LIN {X 0,Y 277.298,Z 529.083,A -85,B 0,C 180,E1 -17480.317,E2 -17480.317} C_VEL
LIN {X 0,Y 276.413,Z 532.07,A -85,B 0,C 180,E1 -17482.419,E2 -17482.419} C_VEL
LIN {X 0,Y 275.927,Z 533.774,A -85,B 0,C 180,E1 -17484.049,E2 -17484.049} C_VEL
LIN {X 0,Y 275.323,Z 535.445,A -85,B 0,C 180,E1 -17486.689,E2 -17486.689} C_VEL
LIN {X 0,Y 274.975,Z 535.726,A -85,B 0,C 180,E1 -17489.654,E2 -17489.654} C_VEL
LIN {X 0,Y 274.909,Z 534.486,A -85,B 0,C 180,E1 -17492.47,E2 -17492.47} C_VEL
LIN {X 0,Y 275.167,Z 531.808,A -85,B 0,C 180,E1 -17495.18,E2 -17495.18} C_VEL
LIN {X 0,Y 275.645,Z 527.856,A -85,B 0,C 180,E1 -17497.774,E2 -17497.774} C_VEL
LIN {X 0,Y 276.168,Z 522.667,A -85,B 0,C 180,E1 -17500.227,E2 -17500.227} C_VEL
LIN {X 0,Y 277.018,Z 516.038,A -85,B 0,C 180,E1 -17502.627,E2 -17502.627} C_VEL
LIN {X 0,Y 278.075,Z 507.892,A -85,B 0,C 180,E1 -17504.952,E2 -17504.952} C_VEL
LIN {X 0,Y 279.237,Z 499.452,A -85,B 0,C 180,E1 -17506.876,E2 -17506.876} C_VEL
LIN {X 0,Y 280.566,Z 489.56,A -85,B 0,C 180,E1 -17508.718,E2 -17508.718} C_VEL
LIN {X 0,Y 282.003,Z 478.351,A -85,B 0,C 180,E1 -17510.385,E2 -17510.385} C_VEL
LIN {X 0,Y 283.262,Z 466.509,A -85,B 0,C 180,E1 -17511.785,E2 -17511.785} C_VEL
LIN {X 0,Y 281.61,Z 454.332,A -85,B 0,C 180,E1 -17513.056,E2 -17513.056} C_VEL
LIN {X 0,Y 279.109,Z 440.408,A -85,B 0,C 180,E1 -17514.219,E2 -17514.219} C_VEL
LIN {X 0,Y 276.812,Z 428.738,A -85,B 0,C 180,E1 -17514.965,E2 -17514.965} C_VEL
LIN {X 0,Y 277.178,Z 422.689,A -85,B 0,C 180,E1 -17518.68,E2 -17518.68} C_VEL
LIN {X 0,Y 277.552,Z 416.666,A -85,B 0,C 180,E1 -17522.404,E2 -17522.404} C_VEL
LIN {X 0,Y 277.936,Z 410.649,A -85,B 0,C 180,E1 -17526.132,E2 -17526.132} C_VEL
LIN {X 0,Y 277.632,Z 407.009,A -85,B 0,C 180,E1 -17528.463,E2 -17528.463} C_VEL
LIN {X 0,Y 277.421,Z 405.931,A -85,B 0,C 180,E1 -17529.224,E2 -17529.224} C_VEL
LIN {X 0,Y 277.446,Z 405.925,A -85,B 0,C 180,E1 -17534.275,E2 -17534.275} C_VEL
LIN {X 0,Y 277.436,Z 405.93,A -85,B 0,C 180,E1 -17538.305,E2 -17538.305} C_VEL
LIN {X 0,Y 277.571,Z 405.911,A -85,B 0,C 180,E1 -17541.259,E2 -17541.259} C_VEL
LIN {X 0,Y 277.511,Z 405.956,A -85,B 0,C 180,E1 -17544.73,E2 -17544.73} C_VEL
LIN {X 0,Y 278.433,Z 410.139,A -85,B 0,C 180,E1 -17548.55,E2 -17548.55} C_VEL
LIN {X 0,Y 278.074,Z 413.616,A -85,B 0,C 180,E1 -17551.445,E2 -17551.445} C_VEL
LIN {X 0,Y 277.432,Z 418.956,A -85,B 0,C 180,E1 -17555.812,E2 -17555.812} C_VEL
LIN {X 0,Y 277.034,Z 422.666,A -85,B 0,C 180,E1 -17558.752,E2 -17558.752} C_VEL
LIN {X 0,Y 276.611,Z 427.071,A -85,B 0,C 180,E1 -17562.189,E2 -17562.189} C_VEL
LIN {X 0,Y 279.223,Z 439.231,A -85,B 0,C 180,E1 -17563.089,E2 -17563.089} C_VEL
LIN {X 0,Y 281.351,Z 451.494,A -85,B 0,C 180,E1 -17564.277,E2 -17564.277} C_VEL
LIN {X 0,Y 282.477,Z 460.237,A -85,B 0,C 180,E1 -17565.325,E2 -17565.325} C_VEL
LIN {X 0,Y 281.293,Z 470.488,A -85,B 0,C 180,E1 -17566.694,E2 -17566.694} C_VEL
LIN {X 0,Y 280.009,Z 480.226,A -85,B 0,C 180,E1 -17568.349,E2 -17568.349} C_VEL
LIN {X 0,Y 278.753,Z 489.099,A -85,B 0,C 180,E1 -17570.28,E2 -17570.28} C_VEL
LIN {X 0,Y 277.708,Z 496.37,A -85,B 0,C 180,E1 -17572.305,E2 -17572.305} C_VEL
LIN {X 0,Y 277.006,Z 501.3,A -85,B 0,C 180,E1 -17574.026,E2 -17574.026} C_VEL
LIN {X 0,Y 276.268,Z 506.386,A -85,B 0,C 180,E1 -17576.303,E2 -17576.303} C_VEL
LIN {X 0,Y 275.857,Z 509.379,A -85,B 0,C 180,E1 -17578.116,E2 -17578.116} C_VEL
LIN {X 0,Y 275.478,Z 512.199,A -85,B 0,C 180,E1 -17580.675,E2 -17580.675} C_VEL
LIN {X 0,Y 275.366,Z 513.344,A -85,B 0,C 180,E1 -17582.624,E2 -17582.624} C_VEL
LIN {X 0,Y 275.417,Z 513.666,A -85,B 0,C 180,E1 -17584.147,E2 -17584.147} C_VEL
LIN {X 0,Y 275.596,Z 513.368,A -85,B 0,C 180,E1 -17585.906,E2 -17585.906} C_VEL
LIN {X 0,Y 275.986,Z 512.222,A -85,B 0,C 180,E1 -17587.87,E2 -17587.87} C_VEL
LIN {X 0,Y 276.777,Z 509.44,A -85,B 0,C 180,E1 -17590.38,E2 -17590.38} C_VEL
LIN {X 0,Y 277.754,Z 505.303,A -85,B 0,C 180,E1 -17592.796,E2 -17592.796} C_VEL
LIN {X 0,Y 279.084,Z 499.564,A -85,B 0,C 180,E1 -17595.163,E2 -17595.163} C_VEL
LIN {X 0,Y 280.373,Z 493.538,A -85,B 0,C 180,E1 -17597.076,E2 -17597.076} C_VEL
LIN {X 0,Y 282.213,Z 485.156,A -85,B 0,C 180,E1 -17599.13,E2 -17599.13} C_VEL
LIN {X 0,Y 283.843,Z 477.123,A -85,B 0,C 180,E1 -17600.686,E2 -17600.686} C_VEL
LIN {X 0,Y 285.699,Z 466.304,A -85,B 0,C 180,E1 -17602.339,E2 -17602.339} C_VEL
LIN {X 0,Y 285.302,Z 460.121,A -85,B 0,C 180,E1 -17603.232,E2 -17603.232} C_VEL
LIN {X 0,Y 283.597,Z 449.539,A -85,B 0,C 180,E1 -17604.624,E2 -17604.624} C_VEL
LIN {X 0,Y 281.033,Z 439.046,A -85,B 0,C 180,E1 -17605.814,E2 -17605.814} C_VEL
LIN {X 0,Y 277.584,Z 428.375,A -85,B 0,C 180,E1 -17606.913,E2 -17606.913} C_VEL
LIN {X 0,Y 278.098,Z 423.388,A -85,B 0,C 180,E1 -17611.305,E2 -17611.305} C_VEL
LIN {X 0,Y 278.623,Z 419.781,A -85,B 0,C 180,E1 -17614.609,E2 -17614.609} C_VEL
LIN {X 0,Y 278.806,Z 416.478,A -85,B 0,C 180,E1 -17617.784,E2 -17617.784} C_VEL
LIN {X 0,Y 278.619,Z 413.529,A -85,B 0,C 180,E1 -17620.858,E2 -17620.858} C_VEL
LIN {X 0,Y 278.253,Z 410.854,A -85,B 0,C 180,E1 -17623.87,E2 -17623.87} C_VEL
LIN {X 0,Y 277.652,Z 407.251,A -85,B 0,C 180,E1 -17628.317,E2 -17628.317} C_VEL
LIN {X 0,Y 277.514,Z 405.917,A -85,B 0,C 180,E1 -17630.153,E2 -17630.153} C_VEL
LIN {X 0,Y 277.631,Z 405.905,A -85,B 0,C 180,E1 -17632.729,E2 -17632.729} C_VEL
LIN {X 0,Y 277.669,Z 405.898,A -85,B 0,C 180,E1 -17636.986,E2 -17636.986} C_VEL
LIN {X 0,Y 277.204,Z 405.963,A -85,B 0,C 180,E1 -17638.198,E2 -17638.198} C_VEL
LIN {X 0,Y 275.718,Z 406.15,A -85,B 0,C 180,E1 -17639.389,E2 -17639.389} C_VEL
LIN {X 0,Y 271.004,Z 406.729,A -85,B 0,C 180,E1 -17642.602,E2 -17642.602} C_VEL
LIN {X 0,Y 270.557,Z 406.778,A -85,B 0,C 180,E1 -17643.444,E2 -17643.444} C_VEL
LIN {X 0,Y 270.591,Z 406.776,A -85,B 0,C 180,E1 -17647.462,E2 -17647.462} C_VEL
LIN {X 0,Y 270.422,Z 406.798,A -85,B 0,C 180,E1 -17650.482,E2 -17650.482} C_VEL
LIN {X 0,Y 270.383,Z 406.8,A -85,B 0,C 180,E1 -17655.066,E2 -17655.066} C_VEL
LIN {X 0,Y 270.308,Z 406.815,A -85,B 0,C 180,E1 -17659.756,E2 -17659.756} C_VEL
LIN {X 0,Y 270.261,Z 406.814,A -85,B 0,C 180,E1 -17664.587,E2 -17664.587} C_VEL
LIN {X 0,Y 270.255,Z 406.817,A -85,B 0,C 180,E1 -17667.911,E2 -17667.911} C_VEL
LIN {X 0,Y 270.168,Z 406.831,A -85,B 0,C 180,E1 -17671.351,E2 -17671.351} C_VEL
LIN {X 0,Y 270.265,Z 407.011,A -85,B 0,C 180,E1 -17675.618,E2 -17675.618} C_VEL
LIN {X 0,Y 270.839,Z 409.72,A -85,B 0,C 180,E1 -17678.886,E2 -17678.886} C_VEL
LIN {X 0,Y 271.495,Z 412.982,A -85,B 0,C 180,E1 -17682.303,E2 -17682.303} C_VEL
LIN {X 0,Y 272.353,Z 416.818,A -85,B 0,C 180,E1 -17685.841,E2 -17685.841} C_VEL
LIN {X 0,Y 273.431,Z 422.485,A -85,B 0,C 180,E1 -17690.453,E2 -17690.453} C_VEL
LIN {X 0,Y 274.584,Z 428.793,A -85,B 0,C 180,E1 -17694.99,E2 -17694.99} C_VEL
LIN {X 0,Y 274.945,Z 431.299,A -85,B 0,C 180,E1 -17696.667,E2 -17696.667} C_VEL
LIN {X 0,Y 274.499,Z 434.05,A -85,B 0,C 180,E1 -17698.351,E2 -17698.351} C_VEL
LIN {X 0,Y 272.629,Z 441.637,A -85,B 0,C 180,E1 -17702.68,E2 -17702.68} C_VEL
LIN {X 0,Y 275.821,Z 455.459,A -85,B 0,C 180,E1 -17703.791,E2 -17703.791} C_VEL
LIN {X 0,Y 277.753,Z 468.394,A -85,B 0,C 180,E1 -17705.038,E2 -17705.038} C_VEL
LIN {X 0,Y 278.418,Z 478.611,A -85,B 0,C 180,E1 -17706.183,E2 -17706.183} C_VEL
LIN {X 0,Y 278.3,Z 489.099,A -85,B 0,C 180,E1 -17707.549,E2 -17707.549} C_VEL
LIN {X 0,Y 276.287,Z 499.847,A -85,B 0,C 180,E1 -17709.142,E2 -17709.142} C_VEL
LIN {X 0,Y 274.262,Z 509.481,A -85,B 0,C 180,E1 -17710.934,E2 -17710.934} C_VEL
LIN {X 0,Y 272.621,Z 517.98,A -85,B 0,C 180,E1 -17712.936,E2 -17712.936} C_VEL
LIN {X 0,Y 271.197,Z 524.971,A -85,B 0,C 180,E1 -17714.984,E2 -17714.984} C_VEL
LIN {X 0,Y 269.826,Z 531.068,A -85,B 0,C 180,E1 -17717.213,E2 -17717.213} C_VEL
LIN {X 0,Y 269.001,Z 535.877,A -85,B 0,C 180,E1 -17719.466,E2 -17719.466} C_VEL
LIN {X 0,Y 268.404,Z 540.987,A -85,B 0,C 180,E1 -17722.481,E2 -17722.481} C_VEL
LIN {X 0,Y 268.227,Z 544.686,A -85,B 0,C 180,E1 -17724.668,E2 -17724.668} C_VEL
LIN {X 0,Y 268.229,Z 547.519,A -85,B 0,C 180,E1 -17727,E2 -17727} C_VEL
LIN {X 0,Y 268.234,Z 548.777,A -85,B 0,C 180,E1 -17728.502,E2 -17728.502} C_VEL
LIN {X 0,Y 268.229,Z 549.619,A -85,B 0,C 180,E1 -17730.003,E2 -17730.003} C_VEL
LIN {X 0,Y 268.227,Z 550.004,A -85,B 0,C 180,E1 -17731.505,E2 -17731.505} C_VEL
LIN {X 0,Y 268.208,Z 549.981,A -85,B 0,C 180,E1 -17733.007,E2 -17733.007} C_VEL
LIN {X 0,Y 268.175,Z 549.223,A -85,B 0,C 180,E1 -17735.212,E2 -17735.212} C_VEL
LIN {X 0,Y 268.456,Z 547.489,A -85,B 0,C 180,E1 -17737.525,E2 -17737.525} C_VEL
LIN {X 0,Y 269.002,Z 544.845,A -85,B 0,C 180,E1 -17739.78,E2 -17739.78} C_VEL
LIN {X 0,Y 269.892,Z 541.2,A -85,B 0,C 180,E1 -17742.027,E2 -17742.027} C_VEL
LIN {X 0,Y 271.146,Z 536.498,A -85,B 0,C 180,E1 -17744.258,E2 -17744.258} C_VEL
LIN {X 0,Y 273.181,Z 529.479,A -85,B 0,C 180,E1 -17746.826,E2 -17746.826} C_VEL
LIN {X 0,Y 275.243,Z 521.489,A -85,B 0,C 180,E1 -17749.133,E2 -17749.133} C_VEL
LIN {X 0,Y 277.76,Z 512.629,A -85,B 0,C 180,E1 -17751.137,E2 -17751.137} C_VEL
LIN {X 0,Y 280.193,Z 503.213,A -85,B 0,C 180,E1 -17752.882,E2 -17752.882} C_VEL
LIN {X 0,Y 282.704,Z 492.898,A -85,B 0,C 180,E1 -17754.415,E2 -17754.415} C_VEL
LIN {X 0,Y 283.337,Z 483.957,A -85,B 0,C 180,E1 -17755.679,E2 -17755.679} C_VEL
LIN {X 0,Y 283.169,Z 472.199,A -85,B 0,C 180,E1 -17757.171,E2 -17757.171} C_VEL
LIN {X 0,Y 281.892,Z 460.18,A -85,B 0,C 180,E1 -17758.598,E2 -17758.598} C_VEL
LIN {X 0,Y 279.764,Z 449.124,A -85,B 0,C 180,E1 -17759.832,E2 -17759.832} C_VEL
LIN {X 0,Y 275.311,Z 434.987,A -85,B 0,C 180,E1 -17761.559,E2 -17761.559} C_VEL
LIN {X 0,Y 275.347,Z 431.758,A -85,B 0,C 180,E1 -17762.616,E2 -17762.616} C_VEL
LIN {X 0,Y 274.35,Z 426.033,A -85,B 0,C 180,E1 -17764.94,E2 -17764.94} C_VEL
LIN {X 0,Y 272.837,Z 419.7,A -85,B 0,C 180,E1 -17768.189,E2 -17768.189} C_VEL
LIN {X 0,Y 271.854,Z 414.556,A -85,B 0,C 180,E1 -17771.434,E2 -17771.434} C_VEL
LIN {X 0,Y 271.327,Z 410.842,A -85,B 0,C 180,E1 -17774.379,E2 -17774.379} C_VEL
LIN {X 0,Y 271.135,Z 409.615,A -85,B 0,C 180,E1 -17775.584,E2 -17775.584} C_VEL
LIN {X 0,Y 270.16,Z 406.826,A -85,B 0,C 180,E1 -17779.798,E2 -17779.798} C_VEL
LIN {X 0,Y 270.231,Z 406.823,A -85,B 0,C 180,E1 -17783.733,E2 -17783.733} C_VEL
LIN {X 0,Y 270.21,Z 406.826,A -85,B 0,C 180,E1 -17786.893,E2 -17786.893} C_VEL
LIN {X 0,Y 270.167,Z 406.831,A -85,B 0,C 180,E1 -17790.379,E2 -17790.379} C_VEL
LIN {X 0,Y 270.222,Z 406.993,A -85,B 0,C 180,E1 -17794.587,E2 -17794.587} C_VEL
LIN {X 0,Y 270.989,Z 409.489,A -85,B 0,C 180,E1 -17799.016,E2 -17799.016} C_VEL
LIN {X 0,Y 271.946,Z 412.845,A -85,B 0,C 180,E1 -17803.484,E2 -17803.484} C_VEL
LIN {X 0,Y 272.58,Z 415.707,A -85,B 0,C 180,E1 -17806.582,E2 -17806.582} C_VEL
LIN {X 0,Y 273.223,Z 418.787,A -85,B 0,C 180,E1 -17809.626,E2 -17809.626} C_VEL
LIN {X 0,Y 273.835,Z 422.113,A -85,B 0,C 180,E1 -17812.627,E2 -17812.627} C_VEL
LIN {X 0,Y 274.033,Z 423.867,A -85,B 0,C 180,E1 -17814.111,E2 -17814.111} C_VEL
LIN {X 0,Y 273.835,Z 426.752,A -85,B 0,C 180,E1 -17816.321,E2 -17816.321} C_VEL
LIN {X 0,Y 273.103,Z 430.671,A -85,B 0,C 180,E1 -17819.123,E2 -17819.123} C_VEL
LIN {X 0,Y 274.489,Z 434.354,A -85,B 0,C 180,E1 -17819.67,E2 -17819.67} C_VEL
LIN {X 0,Y 279.094,Z 445.971,A -85,B 0,C 180,E1 -17821.442,E2 -17821.442} C_VEL
LIN {X 0,Y 282.187,Z 456.631,A -85,B 0,C 180,E1 -17823.038,E2 -17823.038} C_VEL
LIN {X 0,Y 284.054,Z 466.96,A -85,B 0,C 180,E1 -17824.576,E2 -17824.576} C_VEL
LIN {X 0,Y 284.871,Z 476.125,A -85,B 0,C 180,E1 -17826.018,E2 -17826.018} C_VEL
LIN {X 0,Y 283.66,Z 482.538,A -85,B 0,C 180,E1 -17826.89,E2 -17826.89} C_VEL
LIN {X 0,Y 281.037,Z 493.447,A -85,B 0,C 180,E1 -17828.629,E2 -17828.629} C_VEL
LIN {X 0,Y 278.405,Z 503.103,A -85,B 0,C 180,E1 -17830.555,E2 -17830.555} C_VEL
LIN {X 0,Y 275.732,Z 512.265,A -85,B 0,C 180,E1 -17832.886,E2 -17832.886} C_VEL
LIN {X 0,Y 273.512,Z 519.589,A -85,B 0,C 180,E1 -17835.27,E2 -17835.27} C_VEL
LIN {X 0,Y 271.838,Z 525.028,A -85,B 0,C 180,E1 -17837.528,E2 -17837.528} C_VEL
LIN {X 0,Y 270.512,Z 529.16,A -85,B 0,C 180,E1 -17839.739,E2 -17839.739} C_VEL
LIN {X 0,Y 269.713,Z 531.578,A -85,B 0,C 180,E1 -17841.395,E2 -17841.395} C_VEL
LIN {X 0,Y 268.897,Z 534.132,A -85,B 0,C 180,E1 -17843.821,E2 -17843.821} C_VEL
LIN {X 0,Y 268.188,Z 535.826,A -85,B 0,C 180,E1 -17846.998,E2 -17846.998} C_VEL
LIN {X 0,Y 267.867,Z 535.803,A -85,B 0,C 180,E1 -17850.02,E2 -17850.02} C_VEL
LIN {X 0,Y 267.814,Z 534.241,A -85,B 0,C 180,E1 -17852.883,E2 -17852.883} C_VEL
LIN {X 0,Y 268.158,Z 531.305,A -85,B 0,C 180,E1 -17855.659,E2 -17855.659} C_VEL
LIN {X 0,Y 268.653,Z 527.044,A -85,B 0,C 180,E1 -17858.294,E2 -17858.294} C_VEL
LIN {X 0,Y 269.213,Z 521.598,A -85,B 0,C 180,E1 -17860.79,E2 -17860.79} C_VEL
LIN {X 0,Y 270.184,Z 514.647,A -85,B 0,C 180,E1 -17863.25,E2 -17863.25} C_VEL
LIN {X 0,Y 271.271,Z 506.161,A -85,B 0,C 180,E1 -17865.609,E2 -17865.609} C_VEL
LIN {X 0,Y 272.617,Z 497.03,A -85,B 0,C 180,E1 -17867.643,E2 -17867.643} C_VEL
LIN {X 0,Y 273.992,Z 486.938,A -85,B 0,C 180,E1 -17869.454,E2 -17869.454} C_VEL
LIN {X 0,Y 275.506,Z 475.358,A -85,B 0,C 180,E1 -17871.124,E2 -17871.124} C_VEL
LIN {X 0,Y 276.317,Z 466.857,A -85,B 0,C 180,E1 -17872.124,E2 -17872.124} C_VEL
LIN {X 0,Y 274.612,Z 454.825,A -85,B 0,C 180,E1 -17873.419,E2 -17873.419} C_VEL
LIN {X 0,Y 272.214,Z 441.187,A -85,B 0,C 180,E1 -17874.587,E2 -17874.587} C_VEL
LIN {X 0,Y 269.81,Z 428.871,A -85,B 0,C 180,E1 -17875.412,E2 -17875.412} C_VEL
LIN {X 0,Y 270.177,Z 422.923,A -85,B 0,C 180,E1 -17879.138,E2 -17879.138} C_VEL
LIN {X 0,Y 270.575,Z 416.82,A -85,B 0,C 180,E1 -17882.961,E2 -17882.961} C_VEL
LIN {X 0,Y 270.937,Z 411.551,A -85,B 0,C 180,E1 -17886.29,E2 -17886.29} C_VEL
LIN {X 0,Y 270.579,Z 407.891,A -85,B 0,C 180,E1 -17888.673,E2 -17888.673} C_VEL
LIN {X 0,Y 270.389,Z 406.806,A -85,B 0,C 180,E1 -17889.534,E2 -17889.534} C_VEL
LIN {X 0,Y 270.384,Z 406.805,A -85,B 0,C 180,E1 -17894.096,E2 -17894.096} C_VEL
LIN {X 0,Y 270.399,Z 406.805,A -85,B 0,C 180,E1 -17897.996,E2 -17897.996} C_VEL
LIN {X 0,Y 270.528,Z 406.789,A -85,B 0,C 180,E1 -17901.029,E2 -17901.029} C_VEL
LIN {X 0,Y 270.491,Z 406.884,A -85,B 0,C 180,E1 -17904.405,E2 -17904.405} C_VEL
LIN {X 0,Y 271.42,Z 411.271,A -85,B 0,C 180,E1 -17908.513,E2 -17908.513} C_VEL
LIN {X 0,Y 271.039,Z 414.754,A -85,B 0,C 180,E1 -17911.482,E2 -17911.482} C_VEL
LIN {X 0,Y 270.383,Z 420.16,A -85,B 0,C 180,E1 -17915.964,E2 -17915.964} C_VEL
LIN {X 0,Y 269.944,Z 423.882,A -85,B 0,C 180,E1 -17918.983,E2 -17918.983} C_VEL
LIN {X 0,Y 269.606,Z 427.292,A -85,B 0,C 180,E1 -17921.699,E2 -17921.699} C_VEL
LIN {X 0,Y 272.374,Z 439.904,A -85,B 0,C 180,E1 -17922.666,E2 -17922.666} C_VEL
LIN {X 0,Y 274.441,Z 452.083,A -85,B 0,C 180,E1 -17923.888,E2 -17923.888} C_VEL
LIN {X 0,Y 275.56,Z 460.769,A -85,B 0,C 180,E1 -17924.961,E2 -17924.961} C_VEL
LIN {X 0,Y 274.392,Z 470.924,A -85,B 0,C 180,E1 -17926.36,E2 -17926.36} C_VEL
LIN {X 0,Y 273.132,Z 480.269,A -85,B 0,C 180,E1 -17927.981,E2 -17927.981} C_VEL
LIN {X 0,Y 271.764,Z 489.503,A -85,B 0,C 180,E1 -17930.035,E2 -17930.035} C_VEL
LIN {X 0,Y 270.685,Z 496.763,A -85,B 0,C 180,E1 -17932.111,E2 -17932.111} C_VEL
LIN {X 0,Y 269.809,Z 502.654,A -85,B 0,C 180,E1 -17934.262,E2 -17934.262} C_VEL
LIN {X 0,Y 269.165,Z 507.019,A -85,B 0,C 180,E1 -17936.347,E2 -17936.347} C_VEL
LIN {X 0,Y 268.632,Z 510.88,A -85,B 0,C 180,E1 -17938.942,E2 -17938.942} C_VEL
LIN {X 0,Y 268.449,Z 512.229,A -85,B 0,C 180,E1 -17940.239,E2 -17940.239} C_VEL
LIN {X 0,Y 268.297,Z 513.881,A -85,B 0,C 180,E1 -17943.047,E2 -17943.047} C_VEL
LIN {X 0,Y 268.494,Z 513.869,A -85,B 0,C 180,E1 -17945.764,E2 -17945.764} C_VEL
LIN {X 0,Y 269.033,Z 512.393,A -85,B 0,C 180,E1 -17948.401,E2 -17948.401} C_VEL
LIN {X 0,Y 269.919,Z 509.449,A -85,B 0,C 180,E1 -17950.968,E2 -17950.968} C_VEL
LIN {X 0,Y 270.986,Z 505.129,A -85,B 0,C 180,E1 -17953.434,E2 -17953.434} C_VEL
LIN {X 0,Y 272.447,Z 499.247,A -85,B 0,C 180,E1 -17955.855,E2 -17955.855} C_VEL
LIN {X 0,Y 274.042,Z 492.168,A -85,B 0,C 180,E1 -17958.043,E2 -17958.043} C_VEL
LIN {X 0,Y 275.787,Z 484.67,A -85,B 0,C 180,E1 -17959.856,E2 -17959.856} C_VEL
LIN {X 0,Y 277.731,Z 475.146,A -85,B 0,C 180,E1 -17961.664,E2 -17961.664} C_VEL
LIN {X 0,Y 279.109,Z 467.553,A -85,B 0,C 180,E1 -17962.821,E2 -17962.821} C_VEL
LIN {X 0,Y 278.725,Z 461.209,A -85,B 0,C 180,E1 -17963.784,E2 -17963.784} C_VEL
LIN {X 0,Y 276.91,Z 449.799,A -85,B 0,C 180,E1 -17965.343,E2 -17965.343} C_VEL
LIN {X 0,Y 274.172,Z 439.214,A -85,B 0,C 180,E1 -17966.618,E2 -17966.618} C_VEL
LIN {X 0,Y 270.673,Z 428.605,A -85,B 0,C 180,E1 -17967.786,E2 -17967.786} C_VEL
LIN {X 0,Y 271.276,Z 423.758,A -85,B 0,C 180,E1 -17972.204,E2 -17972.204} C_VEL
LIN {X 0,Y 271.768,Z 420.211,A -85,B 0,C 180,E1 -17975.559,E2 -17975.559} C_VEL
LIN {X 0,Y 271.879,Z 417.045,A -85,B 0,C 180,E1 -17978.784,E2 -17978.784} C_VEL
LIN {X 0,Y 271.554,Z 414.216,A -85,B 0,C 180,E1 -17981.907,E2 -17981.907} C_VEL
LIN {X 0,Y 271.19,Z 411.64,A -85,B 0,C 180,E1 -17984.981,E2 -17984.981} C_VEL
LIN {X 0,Y 270.813,Z 409.274,A -85,B 0,C 180,E1 -17988.018,E2 -17988.018} C_VEL
LIN {X 0,Y 270.559,Z 406.784,A -85,B 0,C 180,E1 -17991.599,E2 -17991.599} C_VEL
LIN {X 0,Y 270.525,Z 406.786,A -85,B 0,C 180,E1 -17994.036,E2 -17994.036} C_VEL
LIN {X 0,Y 270.773,Z 406.752,A -85,B 0,C 180,E1 -17998.513,E2 -17998.513} C_VEL
LIN {X 0,Y 270.773,Z 406.752,A -85,B 0,C 180,E1 -18001.488,E2 -18001.488} C_VEL
LIN {X 0,Y 270.557,Z 406.778,A -85,B 0,C 180,E1 -18003.444,E2 -18003.444} C_VEL
LIN {X 0,Y 269.762,Z 406.883,A -85,B 0,C 180,E1 -18004.687,E2 -18004.687} C_VEL
LIN {X 0,Y 266.937,Z 407.228,A -85,B 0,C 180,E1 -18006.716,E2 -18006.716} C_VEL
LIN {X 0,Y 263.778,Z 407.624,A -85,B 0,C 180,E1 -18009.209,E2 -18009.209} C_VEL
LIN {X 0,Y 263.41,Z 407.668,A -85,B 0,C 180,E1 -18010.071,E2 -18010.071} C_VEL
LIN {X 0,Y 263.289,Z 407.689,A -85,B 0,C 180,E1 -18013.901,E2 -18013.901} C_VEL
LIN {X 0,Y 263.256,Z 407.694,A -85,B 0,C 180,E1 -18017.078,E2 -18017.078} C_VEL
LIN {X 0,Y 263.25,Z 407.689,A -85,B 0,C 180,E1 -18020.882,E2 -18020.882} C_VEL
LIN {X 0,Y 263.194,Z 407.698,A -85,B 0,C 180,E1 -18025.293,E2 -18025.293} C_VEL
LIN {X 0,Y 263.163,Z 407.703,A -85,B 0,C 180,E1 -18028.732,E2 -18028.732} C_VEL
LIN {X 0,Y 263.176,Z 407.772,A -85,B 0,C 180,E1 -18033.651,E2 -18033.651} C_VEL
LIN {X 0,Y 263.72,Z 410.183,A -85,B 0,C 180,E1 -18036.927,E2 -18036.927} C_VEL
LIN {X 0,Y 264.197,Z 412.514,A -85,B 0,C 180,E1 -18039.676,E2 -18039.676} C_VEL
LIN {X 0,Y 265.217,Z 417.077,A -85,B 0,C 180,E1 -18044.324,E2 -18044.324} C_VEL
LIN {X 0,Y 266.153,Z 422.073,A -85,B 0,C 180,E1 -18048.695,E2 -18048.695} C_VEL
LIN {X 0,Y 267.063,Z 427.304,A -85,B 0,C 180,E1 -18052.757,E2 -18052.757} C_VEL
LIN {X 0,Y 268.009,Z 432.703,A -85,B 0,C 180,E1 -18056.591,E2 -18056.591} C_VEL
LIN {X 0,Y 267.502,Z 435.448,A -85,B 0,C 180,E1 -18058.306,E2 -18058.306} C_VEL
LIN {X 0,Y 265.935,Z 441.367,A -85,B 0,C 180,E1 -18061.783,E2 -18061.783} C_VEL
LIN {X 0,Y 269.287,Z 455.509,A -85,B 0,C 180,E1 -18063.018,E2 -18063.018} C_VEL
LIN {X 0,Y 271.088,Z 467.636,A -85,B 0,C 180,E1 -18064.242,E2 -18064.242} C_VEL
LIN {X 0,Y 271.871,Z 479.08,A -85,B 0,C 180,E1 -18065.573,E2 -18065.573} C_VEL
LIN {X 0,Y 271.717,Z 489.368,A -85,B 0,C 180,E1 -18066.974,E2 -18066.974} C_VEL
LIN {X 0,Y 269.652,Z 499.994,A -85,B 0,C 180,E1 -18068.604,E2 -18068.604} C_VEL
LIN {X 0,Y 267.548,Z 509.532,A -85,B 0,C 180,E1 -18070.436,E2 -18070.436} C_VEL
LIN {X 0,Y 266.008,Z 516.933,A -85,B 0,C 180,E1 -18072.215,E2 -18072.215} C_VEL
LIN {X 0,Y 264.302,Z 524.829,A -85,B 0,C 180,E1 -18074.583,E2 -18074.583} C_VEL
LIN {X 0,Y 262.874,Z 530.874,A -85,B 0,C 180,E1 -18076.869,E2 -18076.869} C_VEL
LIN {X 0,Y 261.981,Z 535.641,A -85,B 0,C 180,E1 -18079.18,E2 -18079.18} C_VEL
LIN {X 0,Y 261.244,Z 541.848,A -85,B 0,C 180,E1 -18083.05,E2 -18083.05} C_VEL
LIN {X 0,Y 261.096,Z 545.371,A -85,B 0,C 180,E1 -18085.372,E2 -18085.372} C_VEL
LIN {X 0,Y 261.138,Z 547.124,A -85,B 0,C 180,E1 -18086.918,E2 -18086.918} C_VEL
LIN {X 0,Y 261.16,Z 548.424,A -85,B 0,C 180,E1 -18088.461,E2 -18088.461} C_VEL
LIN {X 0,Y 261.154,Z 549.313,A -85,B 0,C 180,E1 -18090.003,E2 -18090.003} C_VEL
LIN {X 0,Y 261.152,Z 549.783,A -85,B 0,C 180,E1 -18091.545,E2 -18091.545} C_VEL
LIN {X 0,Y 261.119,Z 549.805,A -85,B 0,C 180,E1 -18093.089,E2 -18093.089} C_VEL
LIN {X 0,Y 261.157,Z 548.667,A -85,B 0,C 180,E1 -18096.183,E2 -18096.183} C_VEL
LIN {X 0,Y 261.39,Z 547.487,A -85,B 0,C 180,E1 -18097.729,E2 -18097.729} C_VEL
LIN {X 0,Y 262.272,Z 543.865,A -85,B 0,C 180,E1 -18100.815,E2 -18100.815} C_VEL
LIN {X 0,Y 263.313,Z 540,A -85,B 0,C 180,E1 -18103.116,E2 -18103.116} C_VEL
LIN {X 0,Y 264.84,Z 535.031,A -85,B 0,C 180,E1 -18105.392,E2 -18105.392} C_VEL
LIN {X 0,Y 266.764,Z 528.835,A -85,B 0,C 180,E1 -18107.639,E2 -18107.639} C_VEL
LIN {X 0,Y 268.868,Z 521.254,A -85,B 0,C 180,E1 -18109.868,E2 -18109.868} C_VEL
LIN {X 0,Y 271.741,Z 511.878,A -85,B 0,C 180,E1 -18112.028,E2 -18112.028} C_VEL
LIN {X 0,Y 274.357,Z 502.363,A -85,B 0,C 180,E1 -18113.797,E2 -18113.797} C_VEL
LIN {X 0,Y 276.582,Z 493.196,A -85,B 0,C 180,E1 -18115.193,E2 -18115.193} C_VEL
LIN {X 0,Y 277.288,Z 482.326,A -85,B 0,C 180,E1 -18116.784,E2 -18116.784} C_VEL
LIN {X 0,Y 277.127,Z 471.099,A -85,B 0,C 180,E1 -18118.264,E2 -18118.264} C_VEL
LIN {X 0,Y 275.58,Z 458.104,A -85,B 0,C 180,E1 -18119.877,E2 -18119.877} C_VEL
LIN {X 0,Y 274.082,Z 450.681,A -85,B 0,C 180,E1 -18120.781,E2 -18120.781} C_VEL
LIN {X 0,Y 270.401,Z 438.698,A -85,B 0,C 180,E1 -18122.316,E2 -18122.316} C_VEL
LIN {X 0,Y 269.117,Z 434.948,A -85,B 0,C 180,E1 -18122.874,E2 -18122.874} C_VEL
LIN {X 0,Y 268.202,Z 429.316,A -85,B 0,C 180,E1 -18125.207,E2 -18125.207} C_VEL
LIN {X 0,Y 266.466,Z 421.675,A -85,B 0,C 180,E1 -18129.275,E2 -18129.275} C_VEL
LIN {X 0,Y 265.665,Z 417.352,A -85,B 0,C 180,E1 -18132.206,E2 -18132.206} C_VEL
LIN {X 0,Y 265.327,Z 414.721,A -85,B 0,C 180,E1 -18134.341,E2 -18134.341} C_VEL
LIN {X 0,Y 264.884,Z 412.911,A -85,B 0,C 180,E1 -18136.382,E2 -18136.382} C_VEL
LIN {X 0,Y 263.985,Z 410.296,A -85,B 0,C 180,E1 -18140.286,E2 -18140.286} C_VEL
LIN {X 0,Y 263.476,Z 408.985,A -85,B 0,C 180,E1 -18144.067,E2 -18144.067} C_VEL
LIN {X 0,Y 263.329,Z 408.727,A -85,B 0,C 180,E1 -18147.738,E2 -18147.738} C_VEL
LIN {X 0,Y 263.52,Z 409.254,A -85,B 0,C 180,E1 -18151.659,E2 -18151.659} C_VEL
LIN {X 0,Y 263.94,Z 410.363,A -85,B 0,C 180,E1 -18154.872,E2 -18154.872} C_VEL
LIN {X 0,Y 264.433,Z 412.145,A -85,B 0,C 180,E1 -18158.474,E2 -18158.474} C_VEL
LIN {X 0,Y 265.242,Z 414.97,A -85,B 0,C 180,E1 -18162.537,E2 -18162.537} C_VEL
LIN {X 0,Y 265.922,Z 418.079,A -85,B 0,C 180,E1 -18166.239,E2 -18166.239} C_VEL
LIN {X 0,Y 266.843,Z 422.657,A -85,B 0,C 180,E1 -18170.907,E2 -18170.907} C_VEL
LIN {X 0,Y 267.322,Z 426.049,A -85,B 0,C 180,E1 -18173.963,E2 -18173.963} C_VEL
LIN {X 0,Y 267.236,Z 427.907,A -85,B 0,C 180,E1 -18175.474,E2 -18175.474} C_VEL
LIN {X 0,Y 266.75,Z 431.106,A -85,B 0,C 180,E1 -18177.763,E2 -18177.763} C_VEL
LIN {X 0,Y 268.131,Z 434.652,A -85,B 0,C 180,E1 -18178.317,E2 -18178.317} C_VEL
LIN {X 0,Y 271.755,Z 443.605,A -85,B 0,C 180,E1 -18179.814,E2 -18179.814} C_VEL
LIN {X 0,Y 275.434,Z 454.99,A -85,B 0,C 180,E1 -18181.665,E2 -18181.665} C_VEL
LIN {X 0,Y 277.81,Z 466.705,A -85,B 0,C 180,E1 -18183.542,E2 -18183.542} C_VEL
LIN {X 0,Y 278.723,Z 477.886,A -85,B 0,C 180,E1 -18185.364,E2 -18185.364} C_VEL
LIN {X 0,Y 277.675,Z 483.123,A -85,B 0,C 180,E1 -18186.117,E2 -18186.117} C_VEL
LIN {X 0,Y 274.868,Z 493.984,A -85,B 0,C 180,E1 -18187.899,E2 -18187.899} C_VEL
LIN {X 0,Y 272.058,Z 503.705,A -85,B 0,C 180,E1 -18189.899,E2 -18189.899} C_VEL
LIN {X 0,Y 269.451,Z 512.01,A -85,B 0,C 180,E1 -18192.043,E2 -18192.043} C_VEL
LIN {X 0,Y 267.138,Z 519.414,A -85,B 0,C 180,E1 -18194.472,E2 -18194.472} C_VEL
LIN {X 0,Y 264.928,Z 525.857,A -85,B 0,C 180,E1 -18197.246,E2 -18197.246} C_VEL
LIN {X 0,Y 263.553,Z 529.77,A -85,B 0,C 180,E1 -18199.47,E2 -18199.47} C_VEL
LIN {X 0,Y 262.381,Z 533.06,A -85,B 0,C 180,E1 -18202.024,E2 -18202.024} C_VEL
LIN {X 0,Y 261.721,Z 534.821,A -85,B 0,C 180,E1 -18204.071,E2 -18204.071} C_VEL
LIN {X 0,Y 261.359,Z 535.625,A -85,B 0,C 180,E1 -18205.482,E2 -18205.482} C_VEL
LIN {X 0,Y 261.041,Z 536.176,A -85,B 0,C 180,E1 -18207.315,E2 -18207.315} C_VEL
LIN {X 0,Y 260.738,Z 535.796,A -85,B 0,C 180,E1 -18210.393,E2 -18210.393} C_VEL
LIN {X 0,Y 260.778,Z 533.956,A -85,B 0,C 180,E1 -18213.333,E2 -18213.333} C_VEL
LIN {X 0,Y 261.181,Z 530.498,A -85,B 0,C 180,E1 -18216.297,E2 -18216.297} C_VEL
LIN {X 0,Y 261.667,Z 526.206,A -85,B 0,C 180,E1 -18218.836,E2 -18218.836} C_VEL
LIN {X 0,Y 262.338,Z 520.426,A -85,B 0,C 180,E1 -18221.396,E2 -18221.396} C_VEL
LIN {X 0,Y 263.339,Z 513.023,A -85,B 0,C 180,E1 -18223.938,E2 -18223.938} C_VEL
LIN {X 0,Y 264.554,Z 504.259,A -85,B 0,C 180,E1 -18226.311,E2 -18226.311} C_VEL
LIN {X 0,Y 266.138,Z 493.764,A -85,B 0,C 180,E1 -18228.561,E2 -18228.561} C_VEL
LIN {X 0,Y 267.64,Z 482.547,A -85,B 0,C 180,E1 -18230.46,E2 -18230.46} C_VEL
LIN {X 0,Y 269.22,Z 470.499,A -85,B 0,C 180,E1 -18232.072,E2 -18232.072} C_VEL
LIN {X 0,Y 269.287,Z 466.856,A -85,B 0,C 180,E1 -18232.503,E2 -18232.503} C_VEL
LIN {X 0,Y 267.637,Z 455.376,A -85,B 0,C 180,E1 -18233.78,E2 -18233.78} C_VEL
LIN {X 0,Y 265.285,Z 441.809,A -85,B 0,C 180,E1 -18234.987,E2 -18234.987} C_VEL
LIN {X 0,Y 262.841,Z 429.013,A -85,B 0,C 180,E1 -18235.875,E2 -18235.875} C_VEL
LIN {X 0,Y 263.313,Z 421.878,A -85,B 0,C 180,E1 -18240.408,E2 -18240.408} C_VEL
LIN {X 0,Y 263.792,Z 414.785,A -85,B 0,C 180,E1 -18244.935,E2 -18244.935} C_VEL
LIN {X 0,Y 263.893,Z 411.169,A -85,B 0,C 180,E1 -18247.281,E2 -18247.281} C_VEL
LIN {X 0,Y 263.353,Z 407.682,A -85,B 0,C 180,E1 -18249.698,E2 -18249.698} C_VEL
LIN {X 0,Y 263.353,Z 407.681,A -85,B 0,C 180,E1 -18254.519,E2 -18254.519} C_VEL
LIN {X 0,Y 263.356,Z 407.682,A -85,B 0,C 180,E1 -18259.23,E2 -18259.23} C_VEL
LIN {X 0,Y 263.533,Z 407.66,A -85,B 0,C 180,E1 -18262.334,E2 -18262.334} C_VEL
LIN {X 0,Y 263.482,Z 407.785,A -85,B 0,C 180,E1 -18264.064,E2 -18264.064} C_VEL
LIN {X 0,Y 264.407,Z 412.414,A -85,B 0,C 180,E1 -18268.474,E2 -18268.474} C_VEL
LIN {X 0,Y 264.003,Z 415.889,A -85,B 0,C 180,E1 -18271.522,E2 -18271.522} C_VEL
LIN {X 0,Y 263.334,Z 421.326,A -85,B 0,C 180,E1 -18276.125,E2 -18276.125} C_VEL
LIN {X 0,Y 262.865,Z 425.107,A -85,B 0,C 180,E1 -18279.227,E2 -18279.227} C_VEL
LIN {X 0,Y 262.576,Z 427.535,A -85,B 0,C 180,E1 -18281.186,E2 -18281.186} C_VEL
LIN {X 0,Y 265.089,Z 438.671,A -85,B 0,C 180,E1 -18282.047,E2 -18282.047} C_VEL
LIN {X 0,Y 267.025,Z 449.336,A -85,B 0,C 180,E1 -18283.098,E2 -18283.098} C_VEL
LIN {X 0,Y 268.561,Z 460.737,A -85,B 0,C 180,E1 -18284.505,E2 -18284.505} C_VEL
LIN {X 0,Y 268.484,Z 464.092,A -85,B 0,C 180,E1 -18284.957,E2 -18284.957} C_VEL
LIN {X 0,Y 267.124,Z 473.911,A -85,B 0,C 180,E1 -18286.425,E2 -18286.425} C_VEL
LIN {X 0,Y 265.882,Z 483.059,A -85,B 0,C 180,E1 -18288.172,E2 -18288.172} C_VEL
LIN {X 0,Y 264.533,Z 491.477,A -85,B 0,C 180,E1 -18290.201,E2 -18290.201} C_VEL
LIN {X 0,Y 263.493,Z 498.431,A -85,B 0,C 180,E1 -18292.335,E2 -18292.335} C_VEL
LIN {X 0,Y 262.604,Z 503.921,A -85,B 0,C 180,E1 -18294.505,E2 -18294.505} C_VEL
LIN {X 0,Y 261.88,Z 508.884,A -85,B 0,C 180,E1 -18297.139,E2 -18297.139} C_VEL
LIN {X 0,Y 261.54,Z 511.28,A -85,B 0,C 180,E1 -18298.922,E2 -18298.922} C_VEL
LIN {X 0,Y 261.295,Z 513.005,A -85,B 0,C 180,E1 -18300.728,E2 -18300.728} C_VEL
LIN {X 0,Y 261.218,Z 514.369,A -85,B 0,C 180,E1 -18303.484,E2 -18303.484} C_VEL
LIN {X 0,Y 261.496,Z 514.196,A -85,B 0,C 180,E1 -18306.266,E2 -18306.266} C_VEL
LIN {X 0,Y 262.115,Z 512.53,A -85,B 0,C 180,E1 -18308.963,E2 -18308.963} C_VEL
LIN {X 0,Y 263.087,Z 509.468,A -85,B 0,C 180,E1 -18311.585,E2 -18311.585} C_VEL
LIN {X 0,Y 264.261,Z 504.982,A -85,B 0,C 180,E1 -18314.106,E2 -18314.106} C_VEL
LIN {X 0,Y 265.538,Z 500.156,A -85,B 0,C 180,E1 -18316.132,E2 -18316.132} C_VEL
LIN {X 0,Y 267.326,Z 492.723,A -85,B 0,C 180,E1 -18318.52,E2 -18318.52} C_VEL
LIN {X 0,Y 269.408,Z 484.202,A -85,B 0,C 180,E1 -18320.601,E2 -18320.601} C_VEL
LIN {X 0,Y 271.394,Z 474.913,A -85,B 0,C 180,E1 -18322.374,E2 -18322.374} C_VEL
LIN {X 0,Y 272.59,Z 467.932,A -85,B 0,C 180,E1 -18323.462,E2 -18323.462} C_VEL
LIN {X 0,Y 271.626,Z 458.21,A -85,B 0,C 180,E1 -18324.988,E2 -18324.988} C_VEL
LIN {X 0,Y 269.705,Z 447.747,A -85,B 0,C 180,E1 -18326.422,E2 -18326.422} C_VEL
LIN {X 0,Y 266.523,Z 436.825,A -85,B 0,C 180,E1 -18327.782,E2 -18327.782} C_VEL
LIN {X 0,Y 263.758,Z 428.938,A -85,B 0,C 180,E1 -18328.667,E2 -18328.667} C_VEL
LIN {X 0,Y 264.44,Z 424.167,A -85,B 0,C 180,E1 -18333.141,E2 -18333.141} C_VEL
LIN {X 0,Y 264.855,Z 420.751,A -85,B 0,C 180,E1 -18336.546,E2 -18336.546} C_VEL
LIN {X 0,Y 264.944,Z 419.154,A -85,B 0,C 180,E1 -18338.201,E2 -18338.201} C_VEL
LIN {X 0,Y 264.702,Z 416.286,A -85,B 0,C 180,E1 -18341.422,E2 -18341.422} C_VEL
LIN {X 0,Y 264.351,Z 413.665,A -85,B 0,C 180,E1 -18344.583,E2 -18344.583} C_VEL
LIN {X 0,Y 263.827,Z 410.204,A -85,B 0,C 180,E1 -18349.254,E2 -18349.254} C_VEL
LIN {X 0,Y 263.626,Z 408.156,A -85,B 0,C 180,E1 -18352.34,E2 -18352.34} C_VEL
LIN {X 0,Y 263.502,Z 407.662,A -85,B 0,C 180,E1 -18353.492,E2 -18353.492} C_VEL
LIN {X 0,Y 263.738,Z 407.628,A -85,B 0,C 180,E1 -18358.474,E2 -18358.474} C_VEL
LIN {X 0,Y 263.738,Z 407.628,A -85,B 0,C 180,E1 -18361.527,E2 -18361.527} C_VEL
LIN {X 0,Y 263.552,Z 407.654,A -85,B 0,C 180,E1 -18367.663,E2 -18367.663} C_VEL
LIN {X 0,Y 263.41,Z 407.668,A -85,B 0,C 180,E1 -18370.071,E2 -18370.071} C_VEL
LIN {X 0,Y 262.657,Z 407.768,A -85,B 0,C 180,E1 -18371.346,E2 -18371.346} C_VEL
LIN {X 0,Y 259.784,Z 408.124,A -85,B 0,C 180,E1 -18373.424,E2 -18373.424} C_VEL
LIN {X 0,Y 257.378,Z 408.42,A -85,B 0,C 180,E1 -18375.115,E2 -18375.115} C_VEL
LIN {X 0,Y 256.321,Z 408.553,A -85,B 0,C 180,E1 -18376.425,E2 -18376.425} C_VEL
LIN {X 0,Y 256.219,Z 408.564,A -85,B 0,C 180,E1 -18376.869,E2 -18376.869} C_VEL
LIN {X 0,Y 256.185,Z 408.567,A -85,B 0,C 180,E1 -18381.149,E2 -18381.149} C_VEL
LIN {X 0,Y 256.173,Z 408.571,A -85,B 0,C 180,E1 -18385.142,E2 -18385.142} C_VEL
LIN {X 0,Y 256.097,Z 408.577,A -85,B 0,C 180,E1 -18389.602,E2 -18389.602} C_VEL
LIN {X 0,Y 256.105,Z 408.775,A -85,B 0,C 180,E1 -18391.721,E2 -18391.721} C_VEL
LIN {X 0,Y 256.631,Z 410.99,A -85,B 0,C 180,E1 -18395.107,E2 -18395.107} C_VEL
LIN {X 0,Y 257.28,Z 413.978,A -85,B 0,C 180,E1 -18398.924,E2 -18398.924} C_VEL
LIN {X 0,Y 258.288,Z 418.635,A -85,B 0,C 180,E1 -18403.937,E2 -18403.937} C_VEL
LIN {X 0,Y 258.98,Z 422.258,A -85,B 0,C 180,E1 -18407.285,E2 -18407.285} C_VEL
LIN {X 0,Y 259.682,Z 426.101,A -85,B 0,C 180,E1 -18410.511,E2 -18410.511} C_VEL
LIN {X 0,Y 260.696,Z 431.719,A -85,B 0,C 180,E1 -18414.798,E2 -18414.798} C_VEL
LIN {X 0,Y 261.066,Z 434.184,A -85,B 0,C 180,E1 -18416.568,E2 -18416.568} C_VEL
LIN {X 0,Y 260.472,Z 436.852,A -85,B 0,C 180,E1 -18418.26,E2 -18418.26} C_VEL
LIN {X 0,Y 259.269,Z 441.102,A -85,B 0,C 180,E1 -18420.854,E2 -18420.854} C_VEL
LIN {X 0,Y 262.703,Z 455.323,A -85,B 0,C 180,E1 -18422.168,E2 -18422.168} C_VEL
LIN {X 0,Y 264.464,Z 466.796,A -85,B 0,C 180,E1 -18423.374,E2 -18423.374} C_VEL
LIN {X 0,Y 265.312,Z 478.128,A -85,B 0,C 180,E1 -18424.745,E2 -18424.745} C_VEL
LIN {X 0,Y 265.147,Z 489.62,A -85,B 0,C 180,E1 -18426.37,E2 -18426.37} C_VEL
LIN {X 0,Y 263.551,Z 498.012,A -85,B 0,C 180,E1 -18427.671,E2 -18427.671} C_VEL
LIN {X 0,Y 261.26,Z 507.819,A -85,B 0,C 180,E1 -18429.535,E2 -18429.535} C_VEL
LIN {X 0,Y 259.296,Z 516.281,A -85,B 0,C 180,E1 -18431.56,E2 -18431.56} C_VEL
LIN {X 0,Y 257.683,Z 523.605,A -85,B 0,C 180,E1 -18433.77,E2 -18433.77} C_VEL
LIN {X 0,Y 255.937,Z 530.711,A -85,B 0,C 180,E1 -18436.506,E2 -18436.506} C_VEL
LIN {X 0,Y 254.974,Z 535.417,A -85,B 0,C 180,E1 -18438.879,E2 -18438.879} C_VEL
LIN {X 0,Y 254.411,Z 538.987,A -85,B 0,C 180,E1 -18441.265,E2 -18441.265} C_VEL
LIN {X 0,Y 254.167,Z 541.244,A -85,B 0,C 180,E1 -18442.856,E2 -18442.856} C_VEL
LIN {X 0,Y 254.014,Z 544.873,A -85,B 0,C 180,E1 -18445.242,E2 -18445.242} C_VEL
LIN {X 0,Y 254.051,Z 546.718,A -85,B 0,C 180,E1 -18446.832,E2 -18446.832} C_VEL
LIN {X 0,Y 254.087,Z 548.07,A -85,B 0,C 180,E1 -18448.419,E2 -18448.419} C_VEL
LIN {X 0,Y 254.081,Z 549.004,A -85,B 0,C 180,E1 -18450.004,E2 -18450.004} C_VEL
LIN {X 0,Y 254.079,Z 549.535,A -85,B 0,C 180,E1 -18451.589,E2 -18451.589} C_VEL
LIN {X 0,Y 254.012,Z 549.629,A -85,B 0,C 180,E1 -18453.176,E2 -18453.176} C_VEL
LIN {X 0,Y 254.073,Z 548.589,A -85,B 0,C 180,E1 -18456.356,E2 -18456.356} C_VEL
LIN {X 0,Y 254.343,Z 547.49,A -85,B 0,C 180,E1 -18457.945,E2 -18457.945} C_VEL
LIN {X 0,Y 254.753,Z 545.955,A -85,B 0,C 180,E1 -18459.531,E2 -18459.531} C_VEL
LIN {X 0,Y 255.599,Z 542.872,A -85,B 0,C 180,E1 -18461.904,E2 -18461.904} C_VEL
LIN {X 0,Y 256.811,Z 538.765,A -85,B 0,C 180,E1 -18464.262,E2 -18464.262} C_VEL
LIN {X 0,Y 258.692,Z 533.543,A -85,B 0,C 180,E1 -18466.577,E2 -18466.577} C_VEL
LIN {X 0,Y 261.076,Z 526.018,A -85,B 0,C 180,E1 -18469.209,E2 -18469.209} C_VEL
LIN {X 0,Y 263.178,Z 519.158,A -85,B 0,C 180,E1 -18471.135,E2 -18471.135} C_VEL
LIN {X 0,Y 265.719,Z 511.145,A -85,B 0,C 180,E1 -18472.965,E2 -18472.965} C_VEL
LIN {X 0,Y 268.613,Z 501.54,A -85,B 0,C 180,E1 -18474.751,E2 -18474.751} C_VEL
LIN {X 0,Y 270.545,Z 493.611,A -85,B 0,C 180,E1 -18476.003,E2 -18476.003} C_VEL
LIN {X 0,Y 271.347,Z 481.918,A -85,B 0,C 180,E1 -18477.791,E2 -18477.791} C_VEL
LIN {X 0,Y 271.138,Z 470.705,A -85,B 0,C 180,E1 -18479.339,E2 -18479.339} C_VEL
LIN {X 0,Y 269.809,Z 458.335,A -85,B 0,C 180,E1 -18480.961,E2 -18480.961} C_VEL
LIN {X 0,Y 267.627,Z 448.982,A -85,B 0,C 180,E1 -18482.217,E2 -18482.217} C_VEL
LIN {X 0,Y 264.596,Z 439.368,A -85,B 0,C 180,E1 -18483.59,E2 -18483.59} C_VEL
LIN {X 0,Y 262.469,Z 434.923,A -85,B 0,C 180,E1 -18484.432,E2 -18484.432} C_VEL
LIN {X 0,Y 261.646,Z 430.916,A -85,B 0,C 180,E1 -18486.31,E2 -18486.31} C_VEL
LIN {X 0,Y 260.117,Z 423.719,A -85,B 0,C 180,E1 -18490.428,E2 -18490.428} C_VEL
LIN {X 0,Y 259.348,Z 418.838,A -85,B 0,C 180,E1 -18494.101,E2 -18494.101} C_VEL
LIN {X 0,Y 259.137,Z 417.673,A -85,B 0,C 180,E1 -18495.158,E2 -18495.158} C_VEL
LIN {X 0,Y 258.037,Z 414.631,A -85,B 0,C 180,E1 -18499.18,E2 -18499.18} C_VEL
LIN {X 0,Y 257.542,Z 413.155,A -85,B 0,C 180,E1 -18502.318,E2 -18502.318} C_VEL
LIN {X 0,Y 257.297,Z 412.44,A -85,B 0,C 180,E1 -18505.033,E2 -18505.033} C_VEL
LIN {X 0,Y 257.161,Z 412.214,A -85,B 0,C 180,E1 -18508.717,E2 -18508.717} C_VEL
LIN {X 0,Y 257.317,Z 412.806,A -85,B 0,C 180,E1 -18512.334,E2 -18512.334} C_VEL
LIN {X 0,Y 257.666,Z 414.012,A -85,B 0,C 180,E1 -18515.849,E2 -18515.849} C_VEL
LIN {X 0,Y 258.172,Z 415.703,A -85,B 0,C 180,E1 -18519.274,E2 -18519.274} C_VEL
LIN {X 0,Y 258.782,Z 417.904,A -85,B 0,C 180,E1 -18522.618,E2 -18522.618} C_VEL
LIN {X 0,Y 259.493,Z 421.652,A -85,B 0,C 180,E1 -18527.173,E2 -18527.173} C_VEL
LIN {X 0,Y 260.164,Z 424.946,A -85,B 0,C 180,E1 -18530.672,E2 -18530.672} C_VEL
LIN {X 0,Y 260.604,Z 428.265,A -85,B 0,C 180,E1 -18533.807,E2 -18533.807} C_VEL
LIN {X 0,Y 260.304,Z 431.158,A -85,B 0,C 180,E1 -18536.168,E2 -18536.168} C_VEL
LIN {X 0,Y 261.704,Z 434.661,A -85,B 0,C 180,E1 -18536.788,E2 -18536.788} C_VEL
LIN {X 0,Y 262.609,Z 436.625,A -85,B 0,C 180,E1 -18537.171,E2 -18537.171} C_VEL
LIN {X 0,Y 266.343,Z 446.369,A -85,B 0,C 180,E1 -18538.913,E2 -18538.913} C_VEL
LIN {X 0,Y 269.554,Z 456.731,A -85,B 0,C 180,E1 -18540.743,E2 -18540.743} C_VEL
LIN {X 0,Y 271.605,Z 466.604,A -85,B 0,C 180,E1 -18542.43,E2 -18542.43} C_VEL
LIN {X 0,Y 272.504,Z 476.294,A -85,B 0,C 180,E1 -18544.105,E2 -18544.105} C_VEL
LIN {X 0,Y 272.575,Z 480.293,A -85,B 0,C 180,E1 -18544.806,E2 -18544.806} C_VEL
LIN {X 0,Y 269.809,Z 491.031,A -85,B 0,C 180,E1 -18546.477,E2 -18546.477} C_VEL
LIN {X 0,Y 266.984,Z 500.509,A -85,B 0,C 180,E1 -18548.324,E2 -18548.324} C_VEL
LIN {X 0,Y 264.319,Z 508.754,A -85,B 0,C 180,E1 -18550.317,E2 -18550.317} C_VEL
LIN {X 0,Y 261.597,Z 516.784,A -85,B 0,C 180,E1 -18552.751,E2 -18552.751} C_VEL
LIN {X 0,Y 259.555,Z 522.439,A -85,B 0,C 180,E1 -18554.905,E2 -18554.905} C_VEL
LIN {X 0,Y 257.677,Z 527.639,A -85,B 0,C 180,E1 -18557.458,E2 -18557.458} C_VEL
LIN {X 0,Y 256.146,Z 531.547,A -85,B 0,C 180,E1 -18560.031,E2 -18560.031} C_VEL
LIN {X 0,Y 255.053,Z 534.327,A -85,B 0,C 180,E1 -18562.691,E2 -18562.691} C_VEL
LIN {X 0,Y 254.512,Z 535.544,A -85,B 0,C 180,E1 -18564.469,E2 -18564.469} C_VEL
LIN {X 0,Y 253.883,Z 536.427,A -85,B 0,C 180,E1 -18567.642,E2 -18567.642} C_VEL
LIN {X 0,Y 253.629,Z 535.733,A -85,B 0,C 180,E1 -18570.791,E2 -18570.791} C_VEL
LIN {X 0,Y 253.704,Z 533.564,A -85,B 0,C 180,E1 -18573.789,E2 -18573.789} C_VEL
LIN {X 0,Y 254.134,Z 530.06,A -85,B 0,C 180,E1 -18576.676,E2 -18576.676} C_VEL
LIN {X 0,Y 254.669,Z 525.277,A -85,B 0,C 180,E1 -18579.399,E2 -18579.399} C_VEL
LIN {X 0,Y 255.464,Z 519.19,A -85,B 0,C 180,E1 -18582.027,E2 -18582.027} C_VEL
LIN {X 0,Y 256.231,Z 513.622,A -85,B 0,C 180,E1 -18583.951,E2 -18583.951} C_VEL
LIN {X 0,Y 257.41,Z 505.162,A -85,B 0,C 180,E1 -18586.345,E2 -18586.345} C_VEL
LIN {X 0,Y 258.97,Z 495.255,A -85,B 0,C 180,E1 -18588.563,E2 -18588.563} C_VEL
LIN {X 0,Y 260.322,Z 485.565,A -85,B 0,C 180,E1 -18590.33,E2 -18590.33} C_VEL
LIN {X 0,Y 261.876,Z 474.149,A -85,B 0,C 180,E1 -18591.992,E2 -18591.992} C_VEL
LIN {X 0,Y 262.427,Z 468.408,A -85,B 0,C 180,E1 -18592.702,E2 -18592.702} C_VEL
LIN {X 0,Y 260.855,Z 457.12,A -85,B 0,C 180,E1 -18594.033,E2 -18594.033} C_VEL
LIN {X 0,Y 258.72,Z 444.274,A -85,B 0,C 180,E1 -18595.254,E2 -18595.254} C_VEL
LIN {X 0,Y 256.064,Z 430.696,A -85,B 0,C 180,E1 -18596.238,E2 -18596.238} C_VEL
LIN {X 0,Y 255.835,Z 429.179,A -85,B 0,C 180,E1 -18596.337,E2 -18596.337} C_VEL
LIN {X 0,Y 256.261,Z 422.869,A -85,B 0,C 180,E1 -18600.416,E2 -18600.416} C_VEL
LIN {X 0,Y 256.731,Z 416.418,A -85,B 0,C 180,E1 -18604.604,E2 -18604.604} C_VEL
LIN {X 0,Y 256.87,Z 412.06,A -85,B 0,C 180,E1 -18607.475,E2 -18607.475} C_VEL
LIN {X 0,Y 256.286,Z 408.563,A -85,B 0,C 180,E1 -18609.95,E2 -18609.95} C_VEL
LIN {X 0,Y 256.303,Z 408.559,A -85,B 0,C 180,E1 -18614.082,E2 -18614.082} C_VEL
LIN {X 0,Y 256.298,Z 408.561,A -85,B 0,C 180,E1 -18618.93,E2 -18618.93} C_VEL
LIN {X 0,Y 256.495,Z 408.537,A -85,B 0,C 180,E1 -18622.122,E2 -18622.122} C_VEL
LIN {X 0,Y 256.461,Z 408.69,A -85,B 0,C 180,E1 -18623.704,E2 -18623.704} C_VEL
LIN {X 0,Y 257.392,Z 413.546,A -85,B 0,C 180,E1 -18628.432,E2 -18628.432} C_VEL
LIN {X 0,Y 256.967,Z 417.055,A -85,B 0,C 180,E1 -18631.564,E2 -18631.564} C_VEL
LIN {X 0,Y 256.261,Z 422.53,A -85,B 0,C 180,E1 -18636.294,E2 -18636.294} C_VEL
LIN {X 0,Y 255.61,Z 427.72,A -85,B 0,C 180,E1 -18640.642,E2 -18640.642} C_VEL
LIN {X 0,Y 258.293,Z 439.758,A -85,B 0,C 180,E1 -18641.613,E2 -18641.613} C_VEL
LIN {X 0,Y 260.391,Z 451.67,A -85,B 0,C 180,E1 -18642.862,E2 -18642.862} C_VEL
LIN {X 0,Y 261.682,Z 461.7,A -85,B 0,C 180,E1 -18644.162,E2 -18644.162} C_VEL
LIN {X 0,Y 261.317,Z 467.071,A -85,B 0,C 180,E1 -18644.921,E2 -18644.921} C_VEL
LIN {X 0,Y 259.904,Z 476.694,A -85,B 0,C 180,E1 -18646.491,E2 -18646.491} C_VEL
LIN {X 0,Y 258.776,Z 484.543,A -85,B 0,C 180,E1 -18648.095,E2 -18648.095} C_VEL
LIN {X 0,Y 257.337,Z 493.398,A -85,B 0,C 180,E1 -18650.374,E2 -18650.374} C_VEL
LIN {X 0,Y 256.278,Z 500.003,A -85,B 0,C 180,E1 -18652.573,E2 -18652.573} C_VEL
LIN {X 0,Y 255.419,Z 505.17,A -85,B 0,C 180,E1 -18654.769,E2 -18654.769} C_VEL
LIN {X 0,Y 254.813,Z 509.254,A -85,B 0,C 180,E1 -18657.056,E2 -18657.056} C_VEL
LIN {X 0,Y 254.298,Z 512.62,A -85,B 0,C 180,E1 -18659.827,E2 -18659.827} C_VEL
LIN {X 0,Y 254.133,Z 514.023,A -85,B 0,C 180,E1 -18661.693,E2 -18661.693} C_VEL
LIN {X 0,Y 254.17,Z 514.831,A -85,B 0,C 180,E1 -18663.951,E2 -18663.951} C_VEL
LIN {X 0,Y 254.315,Z 514.854,A -85,B 0,C 180,E1 -18665.469,E2 -18665.469} C_VEL
LIN {X 0,Y 254.605,Z 514.225,A -85,B 0,C 180,E1 -18667.387,E2 -18667.387} C_VEL
LIN {X 0,Y 255.214,Z 512.682,A -85,B 0,C 180,E1 -18669.552,E2 -18669.552} C_VEL
LIN {X 0,Y 256.256,Z 509.462,A -85,B 0,C 180,E1 -18672.227,E2 -18672.227} C_VEL
LIN {X 0,Y 257.595,Z 504.826,A -85,B 0,C 180,E1 -18674.818,E2 -18674.818} C_VEL
LIN {X 0,Y 259.31,Z 498.551,A -85,B 0,C 180,E1 -18677.347,E2 -18677.347} C_VEL
LIN {X 0,Y 261.035,Z 491.88,A -85,B 0,C 180,E1 -18679.418,E2 -18679.418} C_VEL
LIN {X 0,Y 263.326,Z 482.775,A -85,B 0,C 180,E1 -18681.595,E2 -18681.595} C_VEL
LIN {X 0,Y 265.28,Z 473.866,A -85,B 0,C 180,E1 -18683.257,E2 -18683.257} C_VEL
LIN {X 0,Y 266.043,Z 468.459,A -85,B 0,C 180,E1 -18684.135,E2 -18684.135} C_VEL
LIN {X 0,Y 264.984,Z 458.443,A -85,B 0,C 180,E1 -18685.773,E2 -18685.773} C_VEL
LIN {X 0,Y 263.163,Z 448.628,A -85,B 0,C 180,E1 -18687.178,E2 -18687.178} C_VEL
LIN {X 0,Y 259.956,Z 437.753,A -85,B 0,C 180,E1 -18688.625,E2 -18688.625} C_VEL
LIN {X 0,Y 256.967,Z 429.719,A -85,B 0,C 180,E1 -18689.605,E2 -18689.605} C_VEL
LIN {X 0,Y 256.889,Z 429.152,A -85,B 0,C 180,E1 -18689.708,E2 -18689.708} C_VEL
LIN {X 0,Y 257.615,Z 424.555,A -85,B 0,C 180,E1 -18694.183,E2 -18694.183} C_VEL
LIN {X 0,Y 257.973,Z 421.033,A -85,B 0,C 180,E1 -18697.847,E2 -18697.847} C_VEL
LIN {X 0,Y 257.836,Z 418.373,A -85,B 0,C 180,E1 -18700.908,E2 -18700.908} C_VEL
LIN {X 0,Y 257.503,Z 415.738,A -85,B 0,C 180,E1 -18704.162,E2 -18704.162} C_VEL
LIN {X 0,Y 257.13,Z 413.362,A -85,B 0,C 180,E1 -18707.37,E2 -18707.37} C_VEL
LIN {X 0,Y 256.953,Z 411.189,A -85,B 0,C 180,E1 -18710.555,E2 -18710.555} C_VEL
LIN {X 0,Y 256.609,Z 409.3,A -85,B 0,C 180,E1 -18713.711,E2 -18713.711} C_VEL
LIN {X 0,Y 256.332,Z 408.557,A -85,B 0,C 180,E1 -18715.282,E2 -18715.282} C_VEL
LIN {X 0,Y 256.702,Z 408.505,A -85,B 0,C 180,E1 -18718.432,E2 -18718.432} C_VEL
LIN {X 0,Y 256.702,Z 408.505,A -85,B 0,C 180,E1 -18721.569,E2 -18721.569} C_VEL
LIN {X 0,Y 256.52,Z 408.532,A -85,B 0,C 180,E1 -18727.874,E2 -18727.874} C_VEL
LIN {X 0,Y 256.29,Z 408.562,A -85,B 0,C 180,E1 -18731.067,E2 -18731.067} C_VEL
LIN {X 0,Y 256.28,Z 408.555,A -85,B 0,C 180,E1 -18735.917,E2 -18735.917} C_VEL
LIN {X 0,Y 256.219,Z 408.564,A -85,B 0,C 180,E1 -18736.869,E2 -18736.869} C_VEL
LIN {X 0,Y 255.498,Z 408.656,A -85,B 0,C 180,E1 -18738.181,E2 -18738.181} C_VEL
LIN {X 0,Y 252.601,Z 409.021,A -85,B 0,C 180,E1 -18740.321,E2 -18740.321} C_VEL
LIN {X 0,Y 250.178,Z 409.322,A -85,B 0,C 180,E1 -18742.062,E2 -18742.062} C_VEL
LIN {X 0,Y 249.153,Z 409.447,A -85,B 0,C 180,E1 -18743.413,E2 -18743.413} C_VEL
LIN {X 0,Y 249.075,Z 409.453,A -85,B 0,C 180,E1 -18743.87,E2 -18743.87} C_VEL
LIN {X 0,Y 249.058,Z 409.454,A -85,B 0,C 180,E1 -18746.84,E2 -18746.84} C_VEL
LIN {X 0,Y 249.088,Z 409.507,A -85,B 0,C 180,E1 -18749.005,E2 -18749.005} C_VEL
LIN {X 0,Y 249.458,Z 411.373,A -85,B 0,C 180,E1 -18752.364,E2 -18752.364} C_VEL
LIN {X 0,Y 250.033,Z 413.921,A -85,B 0,C 180,E1 -18756.177,E2 -18756.177} C_VEL
LIN {X 0,Y 250.686,Z 417.105,A -85,B 0,C 180,E1 -18760.152,E2 -18760.152} C_VEL
LIN {X 0,Y 251.543,Z 420.978,A -85,B 0,C 180,E1 -18764.307,E2 -18764.307} C_VEL
LIN {X 0,Y 252.452,Z 425.778,A -85,B 0,C 180,E1 -18768.734,E2 -18768.734} C_VEL
LIN {X 0,Y 253.477,Z 431.63,A -85,B 0,C 180,E1 -18773.521,E2 -18773.521} C_VEL
LIN {X 0,Y 254.103,Z 435.507,A -85,B 0,C 180,E1 -18776.421,E2 -18776.421} C_VEL
LIN {X 0,Y 253.44,Z 438.255,A -85,B 0,C 180,E1 -18778.21,E2 -18778.21} C_VEL
LIN {X 0,Y 252.666,Z 440.892,A -85,B 0,C 180,E1 -18779.879,E2 -18779.879} C_VEL
LIN {X 0,Y 254.414,Z 447.504,A -85,B 0,C 180,E1 -18780.487,E2 -18780.487} C_VEL
LIN {X 0,Y 256.651,Z 457.672,A -85,B 0,C 180,E1 -18781.533,E2 -18781.533} C_VEL
LIN {X 0,Y 258.275,Z 469.417,A -85,B 0,C 180,E1 -18782.867,E2 -18782.867} C_VEL
LIN {X 0,Y 258.866,Z 480.101,A -85,B 0,C 180,E1 -18784.258,E2 -18784.258} C_VEL
LIN {X 0,Y 258.491,Z 491.248,A -85,B 0,C 180,E1 -18785.936,E2 -18785.936} C_VEL
LIN {X 0,Y 256.258,Z 501.38,A -85,B 0,C 180,E1 -18787.638,E2 -18787.638} C_VEL
LIN {X 0,Y 253.787,Z 511.244,A -85,B 0,C 180,E1 -18789.752,E2 -18789.752} C_VEL
LIN {X 0,Y 252.181,Z 518.02,A -85,B 0,C 180,E1 -18791.565,E2 -18791.565} C_VEL
LIN {X 0,Y 250.551,Z 524.627,A -85,B 0,C 180,E1 -18793.714,E2 -18793.714} C_VEL
LIN {X 0,Y 249.015,Z 530.556,A -85,B 0,C 180,E1 -18796.124,E2 -18796.124} C_VEL
LIN {X 0,Y 247.961,Z 535.2,A -85,B 0,C 180,E1 -18798.56,E2 -18798.56} C_VEL
LIN {X 0,Y 247.355,Z 538.716,A -85,B 0,C 180,E1 -18801.013,E2 -18801.013} C_VEL
LIN {X 0,Y 247.111,Z 540.643,A -85,B 0,C 180,E1 -18802.651,E2 -18802.651} C_VEL
LIN {X 0,Y 246.931,Z 544.374,A -85,B 0,C 180,E1 -18805.106,E2 -18805.106} C_VEL
LIN {X 0,Y 246.965,Z 546.277,A -85,B 0,C 180,E1 -18806.741,E2 -18806.741} C_VEL
LIN {X 0,Y 247.015,Z 547.71,A -85,B 0,C 180,E1 -18808.373,E2 -18808.373} C_VEL
LIN {X 0,Y 247.01,Z 548.687,A -85,B 0,C 180,E1 -18810.004,E2 -18810.004} C_VEL
LIN {X 0,Y 247.006,Z 549.263,A -85,B 0,C 180,E1 -18811.634,E2 -18811.634} C_VEL
LIN {X 0,Y 246.909,Z 549.438,A -85,B 0,C 180,E1 -18813.267,E2 -18813.267} C_VEL
LIN {X 0,Y 246.886,Z 549.179,A -85,B 0,C 180,E1 -18814.903,E2 -18814.903} C_VEL
LIN {X 0,Y 247.293,Z 547.466,A -85,B 0,C 180,E1 -18818.173,E2 -18818.173} C_VEL
LIN {X 0,Y 247.721,Z 546.022,A -85,B 0,C 180,E1 -18819.804,E2 -18819.804} C_VEL
LIN {X 0,Y 249.045,Z 541.821,A -85,B 0,C 180,E1 -18823.051,E2 -18823.051} C_VEL
LIN {X 0,Y 250.549,Z 537.501,A -85,B 0,C 180,E1 -18825.458,E2 -18825.458} C_VEL
LIN {X 0,Y 252.935,Z 531.031,A -85,B 0,C 180,E1 -18828.219,E2 -18828.219} C_VEL
LIN {X 0,Y 255.159,Z 524.144,A -85,B 0,C 180,E1 -18830.529,E2 -18830.529} C_VEL
LIN {X 0,Y 258.209,Z 515.501,A -85,B 0,C 180,E1 -18832.825,E2 -18832.825} C_VEL
LIN {X 0,Y 260.955,Z 506.894,A -85,B 0,C 180,E1 -18834.676,E2 -18834.676} C_VEL
LIN {X 0,Y 263.879,Z 497.562,A -85,B 0,C 180,E1 -18836.285,E2 -18836.285} C_VEL
LIN {X 0,Y 265.074,Z 488.809,A -85,B 0,C 180,E1 -18837.727,E2 -18837.727} C_VEL
LIN {X 0,Y 265.58,Z 476.987,A -85,B 0,C 180,E1 -18839.532,E2 -18839.532} C_VEL
LIN {X 0,Y 264.817,Z 464.473,A -85,B 0,C 180,E1 -18841.307,E2 -18841.307} C_VEL
LIN {X 0,Y 263.336,Z 454.951,A -85,B 0,C 180,E1 -18842.645,E2 -18842.645} C_VEL
LIN {X 0,Y 260.324,Z 444.015,A -85,B 0,C 180,E1 -18844.294,E2 -18844.294} C_VEL
LIN {X 0,Y 257.726,Z 438.912,A -85,B 0,C 180,E1 -18845.343,E2 -18845.343} C_VEL
LIN {X 0,Y 255.633,Z 434.883,A -85,B 0,C 180,E1 -18846.247,E2 -18846.247} C_VEL
LIN {X 0,Y 254.09,Z 427.547,A -85,B 0,C 180,E1 -18850.447,E2 -18850.447} C_VEL
LIN {X 0,Y 253.249,Z 422.187,A -85,B 0,C 180,E1 -18854.503,E2 -18854.503} C_VEL
LIN {X 0,Y 252.749,Z 420.487,A -85,B 0,C 180,E1 -18856.303,E2 -18856.303} C_VEL
LIN {X 0,Y 251.853,Z 417.871,A -85,B 0,C 180,E1 -18860.072,E2 -18860.072} C_VEL
LIN {X 0,Y 251.246,Z 416.293,A -85,B 0,C 180,E1 -18864.025,E2 -18864.025} C_VEL
LIN {X 0,Y 251.015,Z 415.734,A -85,B 0,C 180,E1 -18867.861,E2 -18867.861} C_VEL
LIN {X 0,Y 251.013,Z 415.989,A -85,B 0,C 180,E1 -18871.577,E2 -18871.577} C_VEL
LIN {X 0,Y 251.264,Z 416.996,A -85,B 0,C 180,E1 -18875.193,E2 -18875.193} C_VEL
LIN {X 0,Y 251.696,Z 418.527,A -85,B 0,C 180,E1 -18878.715,E2 -18878.715} C_VEL
LIN {X 0,Y 252.238,Z 420.527,A -85,B 0,C 180,E1 -18882.152,E2 -18882.152} C_VEL
LIN {X 0,Y 252.855,Z 423.912,A -85,B 0,C 180,E1 -18886.618,E2 -18886.618} C_VEL
LIN {X 0,Y 253.512,Z 427.308,A -85,B 0,C 180,E1 -18890.425,E2 -18890.425} C_VEL
LIN {X 0,Y 253.909,Z 430.542,A -85,B 0,C 180,E1 -18893.643,E2 -18893.643} C_VEL
LIN {X 0,Y 253.864,Z 431.442,A -85,B 0,C 180,E1 -18894.396,E2 -18894.396} C_VEL
LIN {X 0,Y 255.376,Z 434.919,A -85,B 0,C 180,E1 -18895.128,E2 -18895.128} C_VEL
LIN {X 0,Y 256.469,Z 437.096,A -85,B 0,C 180,E1 -18895.609,E2 -18895.609} C_VEL
LIN {X 0,Y 258.603,Z 442.247,A -85,B 0,C 180,E1 -18896.65,E2 -18896.65} C_VEL
LIN {X 0,Y 262.375,Z 453.374,A -85,B 0,C 180,E1 -18898.788,E2 -18898.788} C_VEL
LIN {X 0,Y 264.944,Z 463.572,A -85,B 0,C 180,E1 -18900.697,E2 -18900.697} C_VEL
LIN {X 0,Y 266.327,Z 474.294,A -85,B 0,C 180,E1 -18902.646,E2 -18902.646} C_VEL
LIN {X 0,Y 266.477,Z 482.467,A -85,B 0,C 180,E1 -18904.159,E2 -18904.159} C_VEL
LIN {X 0,Y 263.371,Z 493.169,A -85,B 0,C 180,E1 -18905.935,E2 -18905.935} C_VEL
LIN {X 0,Y 260.548,Z 502.016,A -85,B 0,C 180,E1 -18907.751,E2 -18907.751} C_VEL
LIN {X 0,Y 257.703,Z 510.258,A -85,B 0,C 180,E1 -18909.839,E2 -18909.839} C_VEL
LIN {X 0,Y 254.875,Z 517.991,A -85,B 0,C 180,E1 -18912.339,E2 -18912.339} C_VEL
LIN {X 0,Y 252.785,Z 523.305,A -85,B 0,C 180,E1 -18914.49,E2 -18914.49} C_VEL
LIN {X 0,Y 250.542,Z 528.998,A -85,B 0,C 180,E1 -18917.488,E2 -18917.488} C_VEL
LIN {X 0,Y 249.159,Z 532.181,A -85,B 0,C 180,E1 -18919.784,E2 -18919.784} C_VEL
LIN {X 0,Y 248.368,Z 534.04,A -85,B 0,C 180,E1 -18921.583,E2 -18921.583} C_VEL
LIN {X 0,Y 247.38,Z 536.024,A -85,B 0,C 180,E1 -18924.611,E2 -18924.611} C_VEL
LIN {X 0,Y 246.731,Z 536.625,A -85,B 0,C 180,E1 -18927.986,E2 -18927.986} C_VEL
LIN {X 0,Y 246.505,Z 535.59,A -85,B 0,C 180,E1 -18931.201,E2 -18931.201} C_VEL
LIN {X 0,Y 246.664,Z 533.126,A -85,B 0,C 180,E1 -18934.278,E2 -18934.278} C_VEL
LIN {X 0,Y 247.134,Z 529.287,A -85,B 0,C 180,E1 -18937.221,E2 -18937.221} C_VEL
LIN {X 0,Y 247.712,Z 524.256,A -85,B 0,C 180,E1 -18939.997,E2 -18939.997} C_VEL
LIN {X 0,Y 248.607,Z 517.714,A -85,B 0,C 180,E1 -18942.723,E2 -18942.723} C_VEL
LIN {X 0,Y 249.703,Z 509.923,A -85,B 0,C 180,E1 -18945.277,E2 -18945.277} C_VEL
LIN {X 0,Y 251.061,Z 501.15,A -85,B 0,C 180,E1 -18947.57,E2 -18947.57} C_VEL
LIN {X 0,Y 252.543,Z 491.398,A -85,B 0,C 180,E1 -18949.624,E2 -18949.624} C_VEL
LIN {X 0,Y 254.08,Z 481.076,A -85,B 0,C 180,E1 -18951.389,E2 -18951.389} C_VEL
LIN {X 0,Y 255.523,Z 469.995,A -85,B 0,C 180,E1 -18952.903,E2 -18952.903} C_VEL
LIN {X 0,Y 253.868,Z 457.282,A -85,B 0,C 180,E1 -18954.451,E2 -18954.451} C_VEL
LIN {X 0,Y 251.708,Z 444.329,A -85,B 0,C 180,E1 -18955.709,E2 -18955.709} C_VEL
LIN {X 0,Y 249.048,Z 430.666,A -85,B 0,C 180,E1 -18956.731,E2 -18956.731} C_VEL
LIN {X 0,Y 248.84,Z 429.325,A -85,B 0,C 180,E1 -18956.821,E2 -18956.821} C_VEL
LIN {X 0,Y 249.348,Z 422.429,A -85,B 0,C 180,E1 -18961.367,E2 -18961.367} C_VEL
LIN {X 0,Y 249.853,Z 415.546,A -85,B 0,C 180,E1 -18965.926,E2 -18965.926} C_VEL
LIN {X 0,Y 249.647,Z 411.737,A -85,B 0,C 180,E1 -18968.529,E2 -18968.529} C_VEL
LIN {X 0,Y 249.218,Z 409.444,A -85,B 0,C 180,E1 -18970.217,E2 -18970.217} C_VEL
LIN {X 0,Y 249.245,Z 409.439,A -85,B 0,C 180,E1 -18973.619,E2 -18973.619} C_VEL
LIN {X 0,Y 249.246,Z 409.44,A -85,B 0,C 180,E1 -18978.613,E2 -18978.613} C_VEL
LIN {X 0,Y 249.439,Z 409.417,A -85,B 0,C 180,E1 -18981.898,E2 -18981.898} C_VEL
LIN {X 0,Y 249.441,Z 409.596,A -85,B 0,C 180,E1 -18983.322,E2 -18983.322} C_VEL
LIN {X 0,Y 250.376,Z 414.67,A -85,B 0,C 180,E1 -18988.388,E2 -18988.388} C_VEL
LIN {X 0,Y 249.907,Z 418.208,A -85,B 0,C 180,E1 -18991.608,E2 -18991.608} C_VEL
LIN {X 0,Y 249.172,Z 423.733,A -85,B 0,C 180,E1 -18996.474,E2 -18996.474} C_VEL
LIN {X 0,Y 248.628,Z 427.885,A -85,B 0,C 180,E1 -19000.056,E2 -19000.056} C_VEL
LIN {X 0,Y 251.48,Z 440.87,A -85,B 0,C 180,E1 -19001.165,E2 -19001.165} C_VEL
LIN {X 0,Y 253.448,Z 452.196,A -85,B 0,C 180,E1 -19002.406,E2 -19002.406} C_VEL
LIN {X 0,Y 254.762,Z 462.269,A -85,B 0,C 180,E1 -19003.761,E2 -19003.761} C_VEL
LIN {X 0,Y 254.583,Z 466.548,A -85,B 0,C 180,E1 -19004.382,E2 -19004.382} C_VEL
LIN {X 0,Y 253.005,Z 477.03,A -85,B 0,C 180,E1 -19006.124,E2 -19006.124} C_VEL
LIN {X 0,Y 251.759,Z 485.33,A -85,B 0,C 180,E1 -19007.879,E2 -19007.879} C_VEL
LIN {X 0,Y 250.353,Z 493.734,A -85,B 0,C 180,E1 -19010.11,E2 -19010.11} C_VEL
LIN {X 0,Y 249.229,Z 500.451,A -85,B 0,C 180,E1 -19012.409,E2 -19012.409} C_VEL
LIN {X 0,Y 248.251,Z 506.495,A -85,B 0,C 180,E1 -19015.124,E2 -19015.124} C_VEL
LIN {X 0,Y 247.727,Z 509.643,A -85,B 0,C 180,E1 -19016.991,E2 -19016.991} C_VEL
LIN {X 0,Y 247.374,Z 512.049,A -85,B 0,C 180,E1 -19018.875,E2 -19018.875} C_VEL
LIN {X 0,Y 247.064,Z 514.24,A -85,B 0,C 180,E1 -19021.42,E2 -19021.42} C_VEL
LIN {X 0,Y 247.119,Z 515.295,A -85,B 0,C 180,E1 -19024.438,E2 -19024.438} C_VEL
LIN {X 0,Y 247.504,Z 514.776,A -85,B 0,C 180,E1 -19027.339,E2 -19027.339} C_VEL
LIN {X 0,Y 248.344,Z 512.826,A -85,B 0,C 180,E1 -19030.175,E2 -19030.175} C_VEL
LIN {X 0,Y 249.483,Z 509.441,A -85,B 0,C 180,E1 -19032.91,E2 -19032.91} C_VEL
LIN {X 0,Y 250.933,Z 504.671,A -85,B 0,C 180,E1 -19035.559,E2 -19035.559} C_VEL
LIN {X 0,Y 252.778,Z 498.272,A -85,B 0,C 180,E1 -19038.144,E2 -19038.144} C_VEL
LIN {X 0,Y 254.477,Z 492.258,A -85,B 0,C 180,E1 -19040.023,E2 -19040.023} C_VEL
LIN {X 0,Y 256.8,Z 483.359,A -85,B 0,C 180,E1 -19042.206,E2 -19042.206} C_VEL
LIN {X 0,Y 258.586,Z 475.838,A -85,B 0,C 180,E1 -19043.674,E2 -19043.674} C_VEL
LIN {X 0,Y 259.561,Z 470.925,A -85,B 0,C 180,E1 -19044.499,E2 -19044.499} C_VEL
LIN {X 0,Y 258.716,Z 461.155,A -85,B 0,C 180,E1 -19046.202,E2 -19046.202} C_VEL
LIN {X 0,Y 257.208,Z 451.875,A -85,B 0,C 180,E1 -19047.642,E2 -19047.642} C_VEL
LIN {X 0,Y 254.579,Z 442.032,A -85,B 0,C 180,E1 -19049.059,E2 -19049.059} C_VEL
LIN {X 0,Y 250.558,Z 431.45,A -85,B 0,C 180,E1 -19050.496,E2 -19050.496} C_VEL
LIN {X 0,Y 250.025,Z 429.474,A -85,B 0,C 180,E1 -19050.724,E2 -19050.724} C_VEL
LIN {X 0,Y 250.776,Z 425.108,A -85,B 0,C 180,E1 -19055.142,E2 -19055.142} C_VEL
LIN {X 0,Y 251.031,Z 421.918,A -85,B 0,C 180,E1 -19058.657,E2 -19058.657} C_VEL
LIN {X 0,Y 250.798,Z 418.907,A -85,B 0,C 180,E1 -19062.304,E2 -19062.304} C_VEL
LIN {X 0,Y 250.497,Z 416.579,A -85,B 0,C 180,E1 -19065.375,E2 -19065.375} C_VEL
LIN {X 0,Y 250.112,Z 413.239,A -85,B 0,C 180,E1 -19070.294,E2 -19070.294} C_VEL
LIN {X 0,Y 249.802,Z 411.354,A -85,B 0,C 180,E1 -19073.539,E2 -19073.539} C_VEL
LIN {X 0,Y 249.551,Z 409.4,A -85,B 0,C 180,E1 -19077.579,E2 -19077.579} C_VEL
LIN {X 0,Y 249.724,Z 409.379,A -85,B 0,C 180,E1 -19080.001,E2 -19080.001} C_VEL
LIN {X 0,Y 249.448,Z 409.408,A -85,B 0,C 180,E1 -19083.231,E2 -19083.231} C_VEL
LIN {X 0,Y 249.461,Z 409.413,A -85,B 0,C 180,E1 -19088.098,E2 -19088.098} C_VEL
LIN {X 0,Y 249.233,Z 409.439,A -85,B 0,C 180,E1 -19091.385,E2 -19091.385} C_VEL
LIN {X 0,Y 249.223,Z 409.436,A -85,B 0,C 180,E1 -19096.38,E2 -19096.38} C_VEL
LIN {X 0,Y 249.121,Z 409.447,A -85,B 0,C 180,E1 -19101.516,E2 -19101.516} C_VEL
LIN {X 0,Y 249.075,Z 409.453,A -85,B 0,C 180,E1 -19103.87,E2 -19103.87} C_VEL
LIN {X 0,Y 248.439,Z 409.65,A -85,B 0,C 180,E1 -19105.219,E2 -19105.219} C_VEL
LIN {X 0,Y 245.696,Z 410.633,A -85,B 0,C 180,E1 -19107.414,E2 -19107.414} C_VEL
LIN {X 0,Y 243.426,Z 411.729,A -85,B 0,C 180,E1 -19109.196,E2 -19109.196} C_VEL
LIN {X 0,Y 242.547,Z 412.57,A -85,B 0,C 180,E1 -19110.574,E2 -19110.574} C_VEL
LIN {X 0,Y 242.526,Z 412.832,A -85,B 0,C 180,E1 -19111.04,E2 -19111.04} C_VEL
LIN {X 0,Y 243.139,Z 415.456,A -85,B 0,C 180,E1 -19115.318,E2 -19115.318} C_VEL
LIN {X 0,Y 243.749,Z 418.533,A -85,B 0,C 180,E1 -19119.371,E2 -19119.371} C_VEL
LIN {X 0,Y 244.687,Z 422.753,A -85,B 0,C 180,E1 -19124.112,E2 -19124.112} C_VEL
LIN {X 0,Y 245.457,Z 426.907,A -85,B 0,C 180,E1 -19128.112,E2 -19128.112} C_VEL
LIN {X 0,Y 246.245,Z 431.594,A -85,B 0,C 180,E1 -19132.141,E2 -19132.141} C_VEL
LIN {X 0,Y 247.026,Z 435.944,A -85,B 0,C 180,E1 -19135.596,E2 -19135.596} C_VEL
LIN {X 0,Y 246.869,Z 438.279,A -85,B 0,C 180,E1 -19137.26,E2 -19137.26} C_VEL
LIN {X 0,Y 246.088,Z 440.635,A -85,B 0,C 180,E1 -19138.802,E2 -19138.802} C_VEL
LIN {X 0,Y 249.588,Z 454.353,A -85,B 0,C 180,E1 -19140.23,E2 -19140.23} C_VEL
LIN {X 0,Y 251.518,Z 466.493,A -85,B 0,C 180,E1 -19141.644,E2 -19141.644} C_VEL
LIN {X 0,Y 252.339,Z 477.868,A -85,B 0,C 180,E1 -19143.145,E2 -19143.145} C_VEL
LIN {X 0,Y 252.206,Z 487.867,A -85,B 0,C 180,E1 -19144.645,E2 -19144.645} C_VEL
LIN {X 0,Y 251.581,Z 493.995,A -85,B 0,C 180,E1 -19145.671,E2 -19145.671} C_VEL
LIN {X 0,Y 248.968,Z 504.482,A -85,B 0,C 180,E1 -19147.604,E2 -19147.604} C_VEL
LIN {X 0,Y 246.72,Z 512.908,A -85,B 0,C 180,E1 -19149.581,E2 -19149.581} C_VEL
LIN {X 0,Y 244.652,Z 521.088,A -85,B 0,C 180,E1 -19152.017,E2 -19152.017} C_VEL
LIN {X 0,Y 243.192,Z 526.638,A -85,B 0,C 180,E1 -19154.07,E2 -19154.07} C_VEL
LIN {X 0,Y 241.616,Z 532.034,A -85,B 0,C 180,E1 -19156.548,E2 -19156.548} C_VEL
LIN {X 0,Y 240.704,Z 536.243,A -85,B 0,C 180,E1 -19159.064,E2 -19159.064} C_VEL
LIN {X 0,Y 240.038,Z 540.158,A -85,B 0,C 180,E1 -19162.433,E2 -19162.433} C_VEL
LIN {X 0,Y 239.881,Z 543.84,A -85,B 0,C 180,E1 -19164.961,E2 -19164.961} C_VEL
LIN {X 0,Y 239.883,Z 545.792,A -85,B 0,C 180,E1 -19166.645,E2 -19166.645} C_VEL
LIN {X 0,Y 239.944,Z 547.314,A -85,B 0,C 180,E1 -19168.325,E2 -19168.325} C_VEL
LIN {X 0,Y 239.94,Z 548.362,A -85,B 0,C 180,E1 -19170.004,E2 -19170.004} C_VEL
LIN {X 0,Y 239.911,Z 548.988,A -85,B 0,C 180,E1 -19171.682,E2 -19171.682} C_VEL
LIN {X 0,Y 239.802,Z 549.083,A -85,B 0,C 180,E1 -19174.818,E2 -19174.818} C_VEL
LIN {X 0,Y 239.96,Z 548.445,A -85,B 0,C 180,E1 -19176.731,E2 -19176.731} C_VEL
LIN {X 0,Y 240.704,Z 546.077,A -85,B 0,C 180,E1 -19180.093,E2 -19180.093} C_VEL
LIN {X 0,Y 241.695,Z 543.219,A -85,B 0,C 180,E1 -19182.6,E2 -19182.6} C_VEL
LIN {X 0,Y 243.069,Z 539.376,A -85,B 0,C 180,E1 -19185.087,E2 -19185.087} C_VEL
LIN {X 0,Y 245.153,Z 534.443,A -85,B 0,C 180,E1 -19187.522,E2 -19187.522} C_VEL
LIN {X 0,Y 247.444,Z 528.36,A -85,B 0,C 180,E1 -19189.931,E2 -19189.931} C_VEL
LIN {X 0,Y 249.617,Z 522.234,A -85,B 0,C 180,E1 -19191.907,E2 -19191.907} C_VEL
LIN {X 0,Y 252.863,Z 513.359,A -85,B 0,C 180,E1 -19194.205,E2 -19194.205} C_VEL
LIN {X 0,Y 255.953,Z 504.31,A -85,B 0,C 180,E1 -19196.064,E2 -19196.064} C_VEL
LIN {X 0,Y 258.421,Z 495.839,A -85,B 0,C 180,E1 -19197.541,E2 -19197.541} C_VEL
LIN {X 0,Y 259.69,Z 483.68,A -85,B 0,C 180,E1 -19199.6,E2 -19199.6} C_VEL
LIN {X 0,Y 259.73,Z 471.854,A -85,B 0,C 180,E1 -19201.425,E2 -19201.425} C_VEL
LIN {X 0,Y 258.801,Z 461.158,A -85,B 0,C 180,E1 -19203.021,E2 -19203.021} C_VEL
LIN {X 0,Y 256.012,Z 448.697,A -85,B 0,C 180,E1 -19205.014,E2 -19205.014} C_VEL
LIN {X 0,Y 253.515,Z 443.448,A -85,B 0,C 180,E1 -19206.159,E2 -19206.159} C_VEL
LIN {X 0,Y 251.402,Z 439.618,A -85,B 0,C 180,E1 -19207.079,E2 -19207.079} C_VEL
LIN {X 0,Y 248.673,Z 434.73,A -85,B 0,C 180,E1 -19208.41,E2 -19208.41} C_VEL
LIN {X 0,Y 247.701,Z 429.409,A -85,B 0,C 180,E1 -19211.824,E2 -19211.824} C_VEL
LIN {X 0,Y 246.981,Z 425.148,A -85,B 0,C 180,E1 -19215.352,E2 -19215.352} C_VEL
LIN {X 0,Y 246.024,Z 422.296,A -85,B 0,C 180,E1 -19218.926,E2 -19218.926} C_VEL
LIN {X 0,Y 245.63,Z 421.085,A -85,B 0,C 180,E1 -19220.989,E2 -19220.989} C_VEL
LIN {X 0,Y 245.014,Z 419.676,A -85,B 0,C 180,E1 -19224.992,E2 -19224.992} C_VEL
LIN {X 0,Y 244.901,Z 419.323,A -85,B 0,C 180,E1 -19226.958,E2 -19226.958} C_VEL
LIN {X 0,Y 244.76,Z 419.321,A -85,B 0,C 180,E1 -19230.781,E2 -19230.781} C_VEL
LIN {X 0,Y 244.917,Z 420.049,A -85,B 0,C 180,E1 -19234.504,E2 -19234.504} C_VEL
LIN {X 0,Y 245.252,Z 421.388,A -85,B 0,C 180,E1 -19238.128,E2 -19238.128} C_VEL
LIN {X 0,Y 245.725,Z 423.242,A -85,B 0,C 180,E1 -19241.662,E2 -19241.662} C_VEL
LIN {X 0,Y 246.122,Z 425.57,A -85,B 0,C 180,E1 -19245.108,E2 -19245.108} C_VEL
LIN {X 0,Y 246.628,Z 428.25,A -85,B 0,C 180,E1 -19248.493,E2 -19248.493} C_VEL
LIN {X 0,Y 247.175,Z 431.843,A -85,B 0,C 180,E1 -19252.289,E2 -19252.289} C_VEL
LIN {X 0,Y 248.917,Z 435.28,A -85,B 0,C 180,E1 -19253.179,E2 -19253.179} C_VEL
LIN {X 0,Y 250.317,Z 437.443,A -85,B 0,C 180,E1 -19253.826,E2 -19253.826} C_VEL
LIN {X 0,Y 252.51,Z 442.462,A -85,B 0,C 180,E1 -19255.008,E2 -19255.008} C_VEL
LIN {X 0,Y 255.566,Z 451.135,A -85,B 0,C 180,E1 -19256.847,E2 -19256.847} C_VEL
LIN {X 0,Y 258.527,Z 462.209,A -85,B 0,C 180,E1 -19259.097,E2 -19259.097} C_VEL
LIN {X 0,Y 260.079,Z 471.528,A -85,B 0,C 180,E1 -19260.929,E2 -19260.929} C_VEL
LIN {X 0,Y 260.581,Z 481.569,A -85,B 0,C 180,E1 -19262.898,E2 -19262.898} C_VEL
LIN {X 0,Y 260.498,Z 484.022,A -85,B 0,C 180,E1 -19263.381,E2 -19263.381} C_VEL
LIN {X 0,Y 257.145,Z 495.019,A -85,B 0,C 180,E1 -19265.292,E2 -19265.292} C_VEL
LIN {X 0,Y 254.016,Z 504.019,A -85,B 0,C 180,E1 -19267.255,E2 -19267.255} C_VEL
LIN {X 0,Y 250.65,Z 512.818,A -85,B 0,C 180,E1 -19269.685,E2 -19269.685} C_VEL
LIN {X 0,Y 247.785,Z 520.183,A -85,B 0,C 180,E1 -19272.282,E2 -19272.282} C_VEL
LIN {X 0,Y 245.278,Z 525.997,A -85,B 0,C 180,E1 -19274.944,E2 -19274.944} C_VEL
LIN {X 0,Y 243.315,Z 530.368,A -85,B 0,C 180,E1 -19277.594,E2 -19277.594} C_VEL
LIN {X 0,Y 241.754,Z 533.7,A -85,B 0,C 180,E1 -19280.416,E2 -19280.416} C_VEL
LIN {X 0,Y 241.003,Z 535.227,A -85,B 0,C 180,E1 -19282.277,E2 -19282.277} C_VEL
LIN {X 0,Y 240.218,Z 536.523,A -85,B 0,C 180,E1 -19284.906,E2 -19284.906} C_VEL
LIN {X 0,Y 239.631,Z 536.785,A -85,B 0,C 180,E1 -19287.985,E2 -19287.985} C_VEL
LIN {X 0,Y 239.457,Z 536.29,A -85,B 0,C 180,E1 -19289.93,E2 -19289.93} C_VEL
LIN {X 0,Y 239.404,Z 535.196,A -85,B 0,C 180,E1 -19291.898,E2 -19291.898} C_VEL
LIN {X 0,Y 239.625,Z 532.592,A -85,B 0,C 180,E1 -19294.789,E2 -19294.789} C_VEL
LIN {X 0,Y 240.178,Z 528.291,A -85,B 0,C 180,E1 -19297.914,E2 -19297.914} C_VEL
LIN {X 0,Y 240.765,Z 523.134,A -85,B 0,C 180,E1 -19300.625,E2 -19300.625} C_VEL
LIN {X 0,Y 241.742,Z 516.385,A -85,B 0,C 180,E1 -19303.377,E2 -19303.377} C_VEL
LIN {X 0,Y 242.716,Z 509.672,A -85,B 0,C 180,E1 -19305.572,E2 -19305.572} C_VEL
LIN {X 0,Y 244.089,Z 501.091,A -85,B 0,C 180,E1 -19307.851,E2 -19307.851} C_VEL
LIN {X 0,Y 245.614,Z 491.179,A -85,B 0,C 180,E1 -19309.984,E2 -19309.984} C_VEL
LIN {X 0,Y 247.215,Z 480.764,A -85,B 0,C 180,E1 -19311.795,E2 -19311.795} C_VEL
LIN {X 0,Y 248.539,Z 470.383,A -85,B 0,C 180,E1 -19313.251,E2 -19313.251} C_VEL
LIN {X 0,Y 246.944,Z 458.09,A -85,B 0,C 180,E1 -19314.805,E2 -19314.805} C_VEL
LIN {X 0,Y 244.789,Z 445.01,A -85,B 0,C 180,E1 -19316.137,E2 -19316.137} C_VEL
LIN {X 0,Y 242.013,Z 430.605,A -85,B 0,C 180,E1 -19317.257,E2 -19317.257} C_VEL
LIN {X 0,Y 241.849,Z 429.434,A -85,B 0,C 180,E1 -19317.359,E2 -19317.359} C_VEL
LIN {X 0,Y 242.316,Z 423.325,A -85,B 0,C 180,E1 -19321.451,E2 -19321.451} C_VEL
LIN {X 0,Y 242.854,Z 416.442,A -85,B 0,C 180,E1 -19326.096,E2 -19326.096} C_VEL
LIN {X 0,Y 242.607,Z 412.61,A -85,B 0,C 180,E1 -19328.767,E2 -19328.767} C_VEL
LIN {X 0,Y 242.154,Z 410.323,A -85,B 0,C 180,E1 -19330.499,E2 -19330.499} C_VEL
LIN {X 0,Y 242.169,Z 410.32,A -85,B 0,C 180,E1 -19334.856,E2 -19334.856} C_VEL
LIN {X 0,Y 242.331,Z 410.301,A -85,B 0,C 180,E1 -19340.417,E2 -19340.417} C_VEL
LIN {X 0,Y 242.388,Z 410.311,A -85,B 0,C 180,E1 -19342.709,E2 -19342.709} C_VEL
LIN {X 0,Y 243.36,Z 415.796,A -85,B 0,C 180,E1 -19348.341,E2 -19348.341} C_VEL
LIN {X 0,Y 242.847,Z 419.351,A -85,B 0,C 180,E1 -19351.655,E2 -19351.655} C_VEL
LIN {X 0,Y 242.087,Z 424.947,A -85,B 0,C 180,E1 -19356.665,E2 -19356.665} C_VEL
LIN {X 0,Y 241.672,Z 428.107,A -85,B 0,C 180,E1 -19359.458,E2 -19359.458} C_VEL
LIN {X 0,Y 244.639,Z 441.732,A -85,B 0,C 180,E1 -19360.672,E2 -19360.672} C_VEL
LIN {X 0,Y 246.622,Z 453.16,A -85,B 0,C 180,E1 -19361.982,E2 -19361.982} C_VEL
LIN {X 0,Y 247.944,Z 463.982,A -85,B 0,C 180,E1 -19363.52,E2 -19363.52} C_VEL
LIN {X 0,Y 246.946,Z 472.384,A -85,B 0,C 180,E1 -19364.837,E2 -19364.837} C_VEL
LIN {X 0,Y 245.443,Z 481.737,A -85,B 0,C 180,E1 -19366.635,E2 -19366.635} C_VEL
LIN {X 0,Y 243.891,Z 490.955,A -85,B 0,C 180,E1 -19368.912,E2 -19368.912} C_VEL
LIN {X 0,Y 242.733,Z 497.855,A -85,B 0,C 180,E1 -19371.089,E2 -19371.089} C_VEL
LIN {X 0,Y 241.655,Z 504.016,A -85,B 0,C 180,E1 -19373.567,E2 -19373.567} C_VEL
LIN {X 0,Y 240.904,Z 508.529,A -85,B 0,C 180,E1 -19375.946,E2 -19375.946} C_VEL
LIN {X 0,Y 240.312,Z 512.232,A -85,B 0,C 180,E1 -19378.676,E2 -19378.676} C_VEL
LIN {X 0,Y 240.153,Z 513.385,A -85,B 0,C 180,E1 -19379.83,E2 -19379.83} C_VEL
LIN {X 0,Y 239.962,Z 514.842,A -85,B 0,C 180,E1 -19381.86,E2 -19381.86} C_VEL
LIN {X 0,Y 240.07,Z 515.731,A -85,B 0,C 180,E1 -19384.947,E2 -19384.947} C_VEL
LIN {X 0,Y 240.568,Z 515.05,A -85,B 0,C 180,E1 -19387.929,E2 -19387.929} C_VEL
LIN {X 0,Y 241.506,Z 512.937,A -85,B 0,C 180,E1 -19390.834,E2 -19390.834} C_VEL
LIN {X 0,Y 242.763,Z 509.442,A -85,B 0,C 180,E1 -19393.636,E2 -19393.636} C_VEL
LIN {X 0,Y 244.345,Z 504.496,A -85,B 0,C 180,E1 -19396.347,E2 -19396.347} C_VEL
LIN {X 0,Y 246.312,Z 497.955,A -85,B 0,C 180,E1 -19398.986,E2 -19398.986} C_VEL
LIN {X 0,Y 248.371,Z 491.101,A -85,B 0,C 180,E1 -19401.084,E2 -19401.084} C_VEL
LIN {X 0,Y 250.561,Z 482.981,A -85,B 0,C 180,E1 -19403.065,E2 -19403.065} C_VEL
LIN {X 0,Y 252.829,Z 473.532,A -85,B 0,C 180,E1 -19404.866,E2 -19404.866} C_VEL
LIN {X 0,Y 252.991,Z 469.958,A -85,B 0,C 180,E1 -19405.528,E2 -19405.528} C_VEL
LIN {X 0,Y 252.066,Z 460.029,A -85,B 0,C 180,E1 -19407.306,E2 -19407.306} C_VEL
LIN {X 0,Y 250.097,Z 450.011,A -85,B 0,C 180,E1 -19408.912,E2 -19408.912} C_VEL
LIN {X 0,Y 247.067,Z 440.08,A -85,B 0,C 180,E1 -19410.414,E2 -19410.414} C_VEL
LIN {X 0,Y 243.277,Z 430.103,A -85,B 0,C 180,E1 -19411.827,E2 -19411.827} C_VEL
LIN {X 0,Y 243.259,Z 429.611,A -85,B 0,C 180,E1 -19412,E2 -19412} C_VEL
LIN {X 0,Y 243.675,Z 427.348,A -85,B 0,C 180,E1 -19414.366,E2 -19414.366} C_VEL
LIN {X 0,Y 244.103,Z 424.058,A -85,B 0,C 180,E1 -19418.02,E2 -19418.02} C_VEL
LIN {X 0,Y 243.931,Z 420.902,A -85,B 0,C 180,E1 -19421.932,E2 -19421.932} C_VEL
LIN {X 0,Y 243.639,Z 418.655,A -85,B 0,C 180,E1 -19424.953,E2 -19424.953} C_VEL
LIN {X 0,Y 243.265,Z 415.305,A -85,B 0,C 180,E1 -19430.018,E2 -19430.018} C_VEL
LIN {X 0,Y 243.009,Z 413.405,A -85,B 0,C 180,E1 -19433.358,E2 -19433.358} C_VEL
LIN {X 0,Y 242.745,Z 411.01,A -85,B 0,C 180,E1 -19438.341,E2 -19438.341} C_VEL
LIN {X 0,Y 242.645,Z 410.255,A -85,B 0,C 180,E1 -19440.83,E2 -19440.83} C_VEL
LIN {X 0,Y 242.415,Z 410.282,A -85,B 0,C 180,E1 -19446.66,E2 -19446.66} C_VEL
LIN {X 0,Y 242.294,Z 410.297,A -85,B 0,C 180,E1 -19450.023,E2 -19450.023} C_VEL
LIN {X 0,Y 242.148,Z 410.315,A -85,B 0,C 180,E1 -19455.143,E2 -19455.143} C_VEL
LIN {X 0,Y 242.071,Z 410.324,A -85,B 0,C 180,E1 -19458.625,E2 -19458.625} C_VEL
LIN {X 0,Y 242.051,Z 410.329,A -85,B 0,C 180,E1 -19462.177,E2 -19462.177} C_VEL
LIN {X 0,Y 242.05,Z 410.377,A -85,B 0,C 180,E1 -19465.841,E2 -19465.841} C_VEL
LIN {X 0,Y 242.409,Z 412.036,A -85,B 0,C 180,E1 -19469.578,E2 -19469.578} C_VEL
LIN {X 0,Y 242.526,Z 412.832,A -85,B 0,C 180,E1 -19471.04,E2 -19471.04} C_VEL
LIN {X 0,Y 242.065,Z 413.826,A -85,B 0,C 180,E1 -19472.409,E2 -19472.409} C_VEL
LIN {X 0,Y 239.602,Z 416.107,A -85,B 0,C 180,E1 -19474.627,E2 -19474.627} C_VEL
LIN {X 0,Y 237.523,Z 418.079,A -85,B 0,C 180,E1 -19476.426,E2 -19476.426} C_VEL
LIN {X 0,Y 236.761,Z 419.395,A -85,B 0,C 180,E1 -19477.821,E2 -19477.821} C_VEL
LIN {X 0,Y 236.773,Z 419.768,A -85,B 0,C 180,E1 -19478.294,E2 -19478.294} C_VEL
LIN {X 0,Y 237.57,Z 423.602,A -85,B 0,C 180,E1 -19482.876,E2 -19482.876} C_VEL
LIN {X 0,Y 238.246,Z 426.767,A -85,B 0,C 180,E1 -19486.208,E2 -19486.208} C_VEL
LIN {X 0,Y 238.917,Z 430.687,A -85,B 0,C 180,E1 -19489.892,E2 -19489.892} C_VEL
LIN {X 0,Y 239.793,Z 435.651,A -85,B 0,C 180,E1 -19494.12,E2 -19494.12} C_VEL
LIN {X 0,Y 240.17,Z 438.341,A -85,B 0,C 180,E1 -19496.227,E2 -19496.227} C_VEL
LIN {X 0,Y 239.613,Z 440.383,A -85,B 0,C 180,E1 -19497.648,E2 -19497.648} C_VEL
LIN {X 0,Y 243.148,Z 454.263,A -85,B 0,C 180,E1 -19499.204,E2 -19499.204} C_VEL
LIN {X 0,Y 245.179,Z 466.555,A -85,B 0,C 180,E1 -19500.724,E2 -19500.724} C_VEL
LIN {X 0,Y 246.005,Z 478.169,A -85,B 0,C 180,E1 -19502.329,E2 -19502.329} C_VEL
LIN {X 0,Y 245.754,Z 488.423,A -85,B 0,C 180,E1 -19503.95,E2 -19503.95} C_VEL
LIN {X 0,Y 245.14,Z 494.324,A -85,B 0,C 180,E1 -19504.989,E2 -19504.989} C_VEL
LIN {X 0,Y 242.435,Z 504.649,A -85,B 0,C 180,E1 -19506.966,E2 -19506.966} C_VEL
LIN {X 0,Y 240.056,Z 512.967,A -85,B 0,C 180,E1 -19508.988,E2 -19508.988} C_VEL
LIN {X 0,Y 237.893,Z 521.074,A -85,B 0,C 180,E1 -19511.488,E2 -19511.488} C_VEL
LIN {X 0,Y 236.35,Z 526.556,A -85,B 0,C 180,E1 -19513.596,E2 -19513.596} C_VEL
LIN {X 0,Y 234.695,Z 531.891,A -85,B 0,C 180,E1 -19516.144,E2 -19516.144} C_VEL
LIN {X 0,Y 233.702,Z 536.03,A -85,B 0,C 180,E1 -19518.732,E2 -19518.732} C_VEL
LIN {X 0,Y 233.109,Z 539.087,A -85,B 0,C 180,E1 -19521.334,E2 -19521.334} C_VEL
LIN {X 0,Y 232.893,Z 540.768,A -85,B 0,C 180,E1 -19523.071,E2 -19523.071} C_VEL
LIN {X 0,Y 232.795,Z 543.591,A -85,B 0,C 180,E1 -19525.047,E2 -19525.047} C_VEL
LIN {X 0,Y 232.875,Z 546.885,A -85,B 0,C 180,E1 -19528.274,E2 -19528.274} C_VEL
LIN {X 0,Y 232.871,Z 548.031,A -85,B 0,C 180,E1 -19530.004,E2 -19530.004} C_VEL
LIN {X 0,Y 232.818,Z 548.711,A -85,B 0,C 180,E1 -19531.734,E2 -19531.734} C_VEL
LIN {X 0,Y 232.734,Z 548.88,A -85,B 0,C 180,E1 -19535.201,E2 -19535.201} C_VEL
LIN {X 0,Y 232.898,Z 548.383,A -85,B 0,C 180,E1 -19536.936,E2 -19536.936} C_VEL
LIN {X 0,Y 233.704,Z 546.133,A -85,B 0,C 180,E1 -19540.399,E2 -19540.399} C_VEL
LIN {X 0,Y 234.763,Z 543.392,A -85,B 0,C 180,E1 -19542.978,E2 -19542.978} C_VEL
LIN {X 0,Y 236.227,Z 539.704,A -85,B 0,C 180,E1 -19545.535,E2 -19545.535} C_VEL
LIN {X 0,Y 238.417,Z 534.942,A -85,B 0,C 180,E1 -19548.034,E2 -19548.034} C_VEL
LIN {X 0,Y 240.815,Z 529.013,A -85,B 0,C 180,E1 -19550.504,E2 -19550.504} C_VEL
LIN {X 0,Y 243.615,Z 521.748,A -85,B 0,C 180,E1 -19552.924,E2 -19552.924} C_VEL
LIN {X 0,Y 247.073,Z 512.883,A -85,B 0,C 180,E1 -19555.26,E2 -19555.26} C_VEL
LIN {X 0,Y 250.44,Z 503.84,A -85,B 0,C 180,E1 -19557.134,E2 -19557.134} C_VEL
LIN {X 0,Y 252.34,Z 497.611,A -85,B 0,C 180,E1 -19558.263,E2 -19558.263} C_VEL
LIN {X 0,Y 253.774,Z 486.841,A -85,B 0,C 180,E1 -19560.201,E2 -19560.201} C_VEL
LIN {X 0,Y 254.295,Z 476.175,A -85,B 0,C 180,E1 -19561.966,E2 -19561.966} C_VEL
LIN {X 0,Y 253.692,Z 464.704,A -85,B 0,C 180,E1 -19563.789,E2 -19563.789} C_VEL
LIN {X 0,Y 251.853,Z 454.329,A -85,B 0,C 180,E1 -19565.566,E2 -19565.566} C_VEL
LIN {X 0,Y 249.932,Z 449.299,A -85,B 0,C 180,E1 -19566.649,E2 -19566.649} C_VEL
LIN {X 0,Y 247.584,Z 444.665,A -85,B 0,C 180,E1 -19567.85,E2 -19567.85} C_VEL
LIN {X 0,Y 244.265,Z 439.035,A -85,B 0,C 180,E1 -19569.49,E2 -19569.49} C_VEL
LIN {X 0,Y 241.949,Z 434.74,A -85,B 0,C 180,E1 -19570.78,E2 -19570.78} C_VEL
LIN {X 0,Y 241.175,Z 430,A -85,B 0,C 180,E1 -19574.381,E2 -19574.381} C_VEL
LIN {X 0,Y 240.533,Z 427.521,A -85,B 0,C 180,E1 -19576.929,E2 -19576.929} C_VEL
LIN {X 0,Y 239.775,Z 425.471,A -85,B 0,C 180,E1 -19579.846,E2 -19579.846} C_VEL
LIN {X 0,Y 239.036,Z 423.599,A -85,B 0,C 180,E1 -19583.982,E2 -19583.982} C_VEL
LIN {X 0,Y 238.647,Z 422.798,A -85,B 0,C 180,E1 -19587.988,E2 -19587.988} C_VEL
LIN {X 0,Y 238.55,Z 422.933,A -85,B 0,C 180,E1 -19592.114,E2 -19592.114} C_VEL
LIN {X 0,Y 238.68,Z 423.796,A -85,B 0,C 180,E1 -19595.902,E2 -19595.902} C_VEL
LIN {X 0,Y 239.091,Z 425.509,A -85,B 0,C 180,E1 -19600.165,E2 -19600.165} C_VEL
LIN {X 0,Y 239.427,Z 427.055,A -85,B 0,C 180,E1 -19602.93,E2 -19602.93} C_VEL
LIN {X 0,Y 239.819,Z 429.439,A -85,B 0,C 180,E1 -19606.441,E2 -19606.441} C_VEL
LIN {X 0,Y 240.305,Z 432.176,A -85,B 0,C 180,E1 -19609.707,E2 -19609.707} C_VEL
LIN {X 0,Y 242.358,Z 435.875,A -85,B 0,C 180,E1 -19610.904,E2 -19610.904} C_VEL
LIN {X 0,Y 243.952,Z 437.875,A -85,B 0,C 180,E1 -19611.717,E2 -19611.717} C_VEL
LIN {X 0,Y 246.013,Z 441.79,A -85,B 0,C 180,E1 -19612.898,E2 -19612.898} C_VEL
LIN {X 0,Y 248.818,Z 448.614,A -85,B 0,C 180,E1 -19614.618,E2 -19614.618} C_VEL
LIN {X 0,Y 251.984,Z 459.812,A -85,B 0,C 180,E1 -19617.099,E2 -19617.099} C_VEL
LIN {X 0,Y 253.895,Z 469.582,A -85,B 0,C 180,E1 -19619.206,E2 -19619.206} C_VEL
LIN {X 0,Y 254.705,Z 479.113,A -85,B 0,C 180,E1 -19621.185,E2 -19621.185} C_VEL
LIN {X 0,Y 254.566,Z 485.676,A -85,B 0,C 180,E1 -19622.571,E2 -19622.571} C_VEL
LIN {X 0,Y 251.335,Z 495.621,A -85,B 0,C 180,E1 -19624.37,E2 -19624.37} C_VEL
LIN {X 0,Y 247.645,Z 505.566,A -85,B 0,C 180,E1 -19626.628,E2 -19626.628} C_VEL
LIN {X 0,Y 244.132,Z 514.152,A -85,B 0,C 180,E1 -19629.11,E2 -19629.11} C_VEL
LIN {X 0,Y 241.102,Z 521.211,A -85,B 0,C 180,E1 -19631.773,E2 -19631.773} C_VEL
LIN {X 0,Y 238.411,Z 527.001,A -85,B 0,C 180,E1 -19634.588,E2 -19634.588} C_VEL
LIN {X 0,Y 236.127,Z 531.711,A -85,B 0,C 180,E1 -19637.734,E2 -19637.734} C_VEL
LIN {X 0,Y 234.342,Z 535.015,A -85,B 0,C 180,E1 -19641.092,E2 -19641.092} C_VEL
LIN {X 0,Y 233.659,Z 536.193,A -85,B 0,C 180,E1 -19643.017,E2 -19643.017} C_VEL
LIN {X 0,Y 233.038,Z 536.921,A -85,B 0,C 180,E1 -19645.205,E2 -19645.205} C_VEL
LIN {X 0,Y 232.678,Z 537.073,A -85,B 0,C 180,E1 -19646.94,E2 -19646.94} C_VEL
LIN {X 0,Y 232.437,Z 536.707,A -85,B 0,C 180,E1 -19648.932,E2 -19648.932} C_VEL
LIN {X 0,Y 232.304,Z 535.08,A -85,B 0,C 180,E1 -19652.098,E2 -19652.098} C_VEL
LIN {X 0,Y 232.585,Z 531.982,A -85,B 0,C 180,E1 -19655.323,E2 -19655.323} C_VEL
LIN {X 0,Y 233.162,Z 527.556,A -85,B 0,C 180,E1 -19658.395,E2 -19658.395} C_VEL
LIN {X 0,Y 233.905,Z 521.752,A -85,B 0,C 180,E1 -19661.377,E2 -19661.377} C_VEL
LIN {X 0,Y 234.908,Z 514.839,A -85,B 0,C 180,E1 -19664.104,E2 -19664.104} C_VEL
LIN {X 0,Y 236.237,Z 506.166,A -85,B 0,C 180,E1 -19666.82,E2 -19666.82} C_VEL
LIN {X 0,Y 237.862,Z 496.421,A -85,B 0,C 180,E1 -19669.222,E2 -19669.222} C_VEL
LIN {X 0,Y 239.542,Z 485.722,A -85,B 0,C 180,E1 -19671.345,E2 -19671.345} C_VEL
LIN {X 0,Y 241.302,Z 473.683,A -85,B 0,C 180,E1 -19673.22,E2 -19673.22} C_VEL
LIN {X 0,Y 241.588,Z 470.563,A -85,B 0,C 180,E1 -19673.646,E2 -19673.646} C_VEL
LIN {X 0,Y 239.89,Z 458.081,A -85,B 0,C 180,E1 -19675.28,E2 -19675.28} C_VEL
LIN {X 0,Y 237.872,Z 445.434,A -85,B 0,C 180,E1 -19676.607,E2 -19676.607} C_VEL
LIN {X 0,Y 235.1,Z 431.03,A -85,B 0,C 180,E1 -19677.76,E2 -19677.76} C_VEL
LIN {X 0,Y 234.844,Z 429.585,A -85,B 0,C 180,E1 -19677.879,E2 -19677.879} C_VEL
LIN {X 0,Y 235.368,Z 422.941,A -85,B 0,C 180,E1 -19682.427,E2 -19682.427} C_VEL
LIN {X 0,Y 235.852,Z 417.335,A -85,B 0,C 180,E1 -19686.276,E2 -19686.276} C_VEL
LIN {X 0,Y 235.725,Z 414.55,A -85,B 0,C 180,E1 -19688.251,E2 -19688.251} C_VEL
LIN {X 0,Y 235.101,Z 411.202,A -85,B 0,C 180,E1 -19690.799,E2 -19690.799} C_VEL
LIN {X 0,Y 235.115,Z 411.198,A -85,B 0,C 180,E1 -19694.39,E2 -19694.39} C_VEL
LIN {X 0,Y 235.216,Z 411.188,A -85,B 0,C 180,E1 -19699.669,E2 -19699.669} C_VEL
LIN {X 0,Y 235.352,Z 411.218,A -85,B 0,C 180,E1 -19702.274,E2 -19702.274} C_VEL
LIN {X 0,Y 236.006,Z 415.285,A -85,B 0,C 180,E1 -19706.582,E2 -19706.582} C_VEL
LIN {X 0,Y 236.347,Z 416.947,A -85,B 0,C 180,E1 -19708.292,E2 -19708.292} C_VEL
LIN {X 0,Y 235.793,Z 420.538,A -85,B 0,C 180,E1 -19711.704,E2 -19711.704} C_VEL
LIN {X 0,Y 235.005,Z 426.145,A -85,B 0,C 180,E1 -19716.866,E2 -19716.866} C_VEL
LIN {X 0,Y 234.733,Z 428.46,A -85,B 0,C 180,E1 -19718.877,E2 -19718.877} C_VEL
LIN {X 0,Y 237.428,Z 440.62,A -85,B 0,C 180,E1 -19719.957,E2 -19719.957} C_VEL
LIN {X 0,Y 239.326,Z 451.037,A -85,B 0,C 180,E1 -19721.144,E2 -19721.144} C_VEL
LIN {X 0,Y 240.773,Z 461.78,A -85,B 0,C 180,E1 -19722.641,E2 -19722.641} C_VEL
LIN {X 0,Y 241.12,Z 465.703,A -85,B 0,C 180,E1 -19723.266,E2 -19723.266} C_VEL
LIN {X 0,Y 239.603,Z 475.72,A -85,B 0,C 180,E1 -19724.951,E2 -19724.951} C_VEL
LIN {X 0,Y 238.289,Z 484.012,A -85,B 0,C 180,E1 -19726.708,E2 -19726.708} C_VEL
LIN {X 0,Y 236.889,Z 491.57,A -85,B 0,C 180,E1 -19728.672,E2 -19728.672} C_VEL
LIN {X 0,Y 235.672,Z 498.546,A -85,B 0,C 180,E1 -19730.964,E2 -19730.964} C_VEL
LIN {X 0,Y 234.605,Z 504.358,A -85,B 0,C 180,E1 -19733.381,E2 -19733.381} C_VEL
LIN {X 0,Y 233.905,Z 508.605,A -85,B 0,C 180,E1 -19735.66,E2 -19735.66} C_VEL
LIN {X 0,Y 233.383,Z 511.665,A -85,B 0,C 180,E1 -19737.819,E2 -19737.819} C_VEL
LIN {X 0,Y 232.938,Z 514.564,A -85,B 0,C 180,E1 -19740.853,E2 -19740.853} C_VEL
LIN {X 0,Y 232.868,Z 515.683,A -85,B 0,C 180,E1 -19742.899,E2 -19742.899} C_VEL
LIN {X 0,Y 233.063,Z 516.129,A -85,B 0,C 180,E1 -19745.494,E2 -19745.494} C_VEL
LIN {X 0,Y 233.649,Z 515.328,A -85,B 0,C 180,E1 -19748.551,E2 -19748.551} C_VEL
LIN {X 0,Y 234.674,Z 513.058,A -85,B 0,C 180,E1 -19751.523,E2 -19751.523} C_VEL
LIN {X 0,Y 236.042,Z 509.443,A -85,B 0,C 180,E1 -19754.392,E2 -19754.392} C_VEL
LIN {X 0,Y 237.797,Z 504.328,A -85,B 0,C 180,E1 -19757.176,E2 -19757.176} C_VEL
LIN {X 0,Y 239.73,Z 498.256,A -85,B 0,C 180,E1 -19759.653,E2 -19759.653} C_VEL
LIN {X 0,Y 242.276,Z 490.259,A -85,B 0,C 180,E1 -19762.121,E2 -19762.121} C_VEL
LIN {X 0,Y 244.686,Z 481.511,A -85,B 0,C 180,E1 -19764.204,E2 -19764.204} C_VEL
LIN {X 0,Y 246.583,Z 473.514,A -85,B 0,C 180,E1 -19765.737,E2 -19765.737} C_VEL
LIN {X 0,Y 245.992,Z 463.822,A -85,B 0,C 180,E1 -19767.612,E2 -19767.612} C_VEL
LIN {X 0,Y 244.543,Z 454.801,A -85,B 0,C 180,E1 -19769.187,E2 -19769.187} C_VEL
LIN {X 0,Y 241.825,Z 444.63,A -85,B 0,C 180,E1 -19770.871,E2 -19770.871} C_VEL
LIN {X 0,Y 237.669,Z 433.404,A -85,B 0,C 180,E1 -19772.63,E2 -19772.63} C_VEL
LIN {X 0,Y 236.488,Z 430.02,A -85,B 0,C 180,E1 -19773.116,E2 -19773.116} C_VEL
LIN {X 0,Y 237.129,Z 426.223,A -85,B 0,C 180,E1 -19777.339,E2 -19777.339} C_VEL
LIN {X 0,Y 237.07,Z 423.333,A -85,B 0,C 180,E1 -19780.968,E2 -19780.968} C_VEL
LIN {X 0,Y 236.792,Z 420.759,A -85,B 0,C 180,E1 -19784.508,E2 -19784.508} C_VEL
LIN {X 0,Y 236.44,Z 417.39,A -85,B 0,C 180,E1 -19789.727,E2 -19789.727} C_VEL
LIN {X 0,Y 236.194,Z 415.47,A -85,B 0,C 180,E1 -19793.165,E2 -19793.165} C_VEL
LIN {X 0,Y 235.945,Z 413.095,A -85,B 0,C 180,E1 -19798.294,E2 -19798.294} C_VEL
LIN {X 0,Y 235.704,Z 411.908,A -85,B 0,C 180,E1 -19801.709,E2 -19801.709} C_VEL
LIN {X 0,Y 235.213,Z 411.187,A -85,B 0,C 180,E1 -19805.143,E2 -19805.143} C_VEL
LIN {X 0,Y 235.385,Z 411.157,A -85,B 0,C 180,E1 -19806.86,E2 -19806.86} C_VEL
LIN {X 0,Y 235.218,Z 411.18,A -85,B 0,C 180,E1 -19810.328,E2 -19810.328} C_VEL
LIN {X 0,Y 235.095,Z 411.193,A -85,B 0,C 180,E1 -19815.608,E2 -19815.608} C_VEL
LIN {X 0,Y 235.015,Z 411.205,A -85,B 0,C 180,E1 -19819.206,E2 -19819.206} C_VEL
LIN {X 0,Y 235.068,Z 411.439,A -85,B 0,C 180,E1 -19822.068,E2 -19822.068} C_VEL
LIN {X 0,Y 235.253,Z 412.224,A -85,B 0,C 180,E1 -19824.724,E2 -19824.724} C_VEL
LIN {X 0,Y 235.692,Z 414.572,A -85,B 0,C 180,E1 -19830.157,E2 -19830.157} C_VEL
LIN {X 0,Y 236.212,Z 417.021,A -85,B 0,C 180,E1 -19834.424,E2 -19834.424} C_VEL
LIN {X 0,Y 236.773,Z 419.768,A -85,B 0,C 180,E1 -19838.294,E2 -19838.294} C_VEL
LIN {X 0,Y 236.391,Z 421.052,A -85,B 0,C 180,E1 -19839.686,E2 -19839.686} C_VEL
LIN {X 0,Y 234.013,Z 423.766,A -85,B 0,C 180,E1 -19841.936,E2 -19841.936} C_VEL
LIN {X 0,Y 231.984,Z 426.088,A -85,B 0,C 180,E1 -19843.761,E2 -19843.761} C_VEL
LIN {X 0,Y 231.265,Z 427.673,A -85,B 0,C 180,E1 -19845.177,E2 -19845.177} C_VEL
LIN {X 0,Y 231.294,Z 428.141,A -85,B 0,C 180,E1 -19845.657,E2 -19845.657} C_VEL
LIN {X 0,Y 231.943,Z 431.776,A -85,B 0,C 180,E1 -19849.246,E2 -19849.246} C_VEL
LIN {X 0,Y 232.822,Z 436.903,A -85,B 0,C 180,E1 -19853.8,E2 -19853.8} C_VEL
LIN {X 0,Y 233.208,Z 439.73,A -85,B 0,C 180,E1 -19856.122,E2 -19856.122} C_VEL
LIN {X 0,Y 233.119,Z 440.332,A -85,B 0,C 180,E1 -19856.439,E2 -19856.439} C_VEL
LIN {X 0,Y 236.396,Z 452.336,A -85,B 0,C 180,E1 -19857.864,E2 -19857.864} C_VEL
LIN {X 0,Y 238.41,Z 463.059,A -85,B 0,C 180,E1 -19859.249,E2 -19859.249} C_VEL
LIN {X 0,Y 239.42,Z 473.079,A -85,B 0,C 180,E1 -19860.652,E2 -19860.652} C_VEL
LIN {X 0,Y 239.62,Z 483.219,A -85,B 0,C 180,E1 -19862.221,E2 -19862.221} C_VEL
LIN {X 0,Y 238.938,Z 493.589,A -85,B 0,C 180,E1 -19864.059,E2 -19864.059} C_VEL
LIN {X 0,Y 236.467,Z 503.02,A -85,B 0,C 180,E1 -19865.884,E2 -19865.884} C_VEL
LIN {X 0,Y 233.9,Z 511.584,A -85,B 0,C 180,E1 -19867.944,E2 -19867.944} C_VEL
LIN {X 0,Y 231.476,Z 519.838,A -85,B 0,C 180,E1 -19870.494,E2 -19870.494} C_VEL
LIN {X 0,Y 229.519,Z 526.475,A -85,B 0,C 180,E1 -19873.093,E2 -19873.093} C_VEL
LIN {X 0,Y 227.793,Z 531.745,A -85,B 0,C 180,E1 -19875.715,E2 -19875.715} C_VEL
LIN {X 0,Y 226.692,Z 535.813,A -85,B 0,C 180,E1 -19878.379,E2 -19878.379} C_VEL
LIN {X 0,Y 226.047,Z 538.811,A -85,B 0,C 180,E1 -19881.061,E2 -19881.061} C_VEL
LIN {X 0,Y 225.818,Z 540.242,A -85,B 0,C 180,E1 -19882.853,E2 -19882.853} C_VEL
LIN {X 0,Y 225.692,Z 544.805,A -85,B 0,C 180,E1 -19886.433,E2 -19886.433} C_VEL
LIN {X 0,Y 225.782,Z 546.435,A -85,B 0,C 180,E1 -19888.22,E2 -19888.22} C_VEL
LIN {X 0,Y 225.804,Z 547.641,A -85,B 0,C 180,E1 -19890.004,E2 -19890.004} C_VEL
LIN {X 0,Y 225.727,Z 548.423,A -85,B 0,C 180,E1 -19891.788,E2 -19891.788} C_VEL
LIN {X 0,Y 225.65,Z 548.709,A -85,B 0,C 180,E1 -19895.365,E2 -19895.365} C_VEL
LIN {X 0,Y 226.171,Z 547.451,A -85,B 0,C 180,E1 -19898.942,E2 -19898.942} C_VEL
LIN {X 0,Y 227.4,Z 544.567,A -85,B 0,C 180,E1 -19902.498,E2 -19902.498} C_VEL
LIN {X 0,Y 228.824,Z 541.337,A -85,B 0,C 180,E1 -19905.137,E2 -19905.137} C_VEL
LIN {X 0,Y 230.897,Z 537.084,A -85,B 0,C 180,E1 -19907.724,E2 -19907.724} C_VEL
LIN {X 0,Y 233.781,Z 530.747,A -85,B 0,C 180,E1 -19910.689,E2 -19910.689} C_VEL
LIN {X 0,Y 236.631,Z 523.983,A -85,B 0,C 180,E1 -19913.178,E2 -19913.178} C_VEL
LIN {X 0,Y 240.178,Z 515.629,A -85,B 0,C 180,E1 -19915.573,E2 -19915.573} C_VEL
LIN {X 0,Y 243.487,Z 507.222,A -85,B 0,C 180,E1 -19917.508,E2 -19917.508} C_VEL
LIN {X 0,Y 246.307,Z 499.337,A -85,B 0,C 180,E1 -19919.02,E2 -19919.02} C_VEL
LIN {X 0,Y 248.135,Z 488.055,A -85,B 0,C 180,E1 -19921.175,E2 -19921.175} C_VEL
LIN {X 0,Y 248.811,Z 476.912,A -85,B 0,C 180,E1 -19923.119,E2 -19923.119} C_VEL
LIN {X 0,Y 248.667,Z 468.375,A -85,B 0,C 180,E1 -19924.567,E2 -19924.567} C_VEL
LIN {X 0,Y 247.258,Z 458.502,A -85,B 0,C 180,E1 -19926.358,E2 -19926.358} C_VEL
LIN {X 0,Y 246.414,Z 455.528,A -85,B 0,C 180,E1 -19927.003,E2 -19927.003} C_VEL
LIN {X 0,Y 242.738,Z 447.932,A -85,B 0,C 180,E1 -19929.131,E2 -19929.131} C_VEL
LIN {X 0,Y 240.764,Z 444.339,A -85,B 0,C 180,E1 -19930.273,E2 -19930.273} C_VEL
LIN {X 0,Y 238.333,Z 439.879,A -85,B 0,C 180,E1 -19931.739,E2 -19931.739} C_VEL
LIN {X 0,Y 235.222,Z 434.493,A -85,B 0,C 180,E1 -19933.82,E2 -19933.82} C_VEL
LIN {X 0,Y 234.644,Z 431.72,A -85,B 0,C 180,E1 -19936.457,E2 -19936.457} C_VEL
LIN {X 0,Y 234.009,Z 430.002,A -85,B 0,C 180,E1 -19938.666,E2 -19938.666} C_VEL
LIN {X 0,Y 233.123,Z 427.638,A -85,B 0,C 180,E1 -19942.918,E2 -19942.918} C_VEL
LIN {X 0,Y 232.552,Z 426.489,A -85,B 0,C 180,E1 -19947.044,E2 -19947.044} C_VEL
LIN {X 0,Y 232.346,Z 426.276,A -85,B 0,C 180,E1 -19951.054,E2 -19951.054} C_VEL
LIN {X 0,Y 232.375,Z 426.895,A -85,B 0,C 180,E1 -19955.144,E2 -19955.144} C_VEL
LIN {X 0,Y 232.677,Z 428.344,A -85,B 0,C 180,E1 -19959.455,E2 -19959.455} C_VEL
LIN {X 0,Y 232.962,Z 429.81,A -85,B 0,C 180,E1 -19962.441,E2 -19962.441} C_VEL
LIN {X 0,Y 233.386,Z 432.444,A -85,B 0,C 180,E1 -19966.448,E2 -19966.448} C_VEL
LIN {X 0,Y 235.418,Z 436.061,A -85,B 0,C 180,E1 -19967.937,E2 -19967.937} C_VEL
LIN {X 0,Y 237.534,Z 438.647,A -85,B 0,C 180,E1 -19969.24,E2 -19969.24} C_VEL
LIN {X 0,Y 239.483,Z 442.213,A -85,B 0,C 180,E1 -19970.533,E2 -19970.533} C_VEL
LIN {X 0,Y 240.581,Z 443.887,A -85,B 0,C 180,E1 -19971.177,E2 -19971.177} C_VEL
LIN {X 0,Y 243.013,Z 449.135,A -85,B 0,C 180,E1 -19972.81,E2 -19972.81} C_VEL
LIN {X 0,Y 245.204,Z 455.898,A -85,B 0,C 180,E1 -19974.539,E2 -19974.539} C_VEL
LIN {X 0,Y 247.633,Z 467.055,A -85,B 0,C 180,E1 -19977.153,E2 -19977.153} C_VEL
LIN {X 0,Y 248.757,Z 476.045,A -85,B 0,C 180,E1 -19979.19,E2 -19979.19} C_VEL
LIN {X 0,Y 248.882,Z 485.11,A -85,B 0,C 180,E1 -19981.213,E2 -19981.213} C_VEL
LIN {X 0,Y 248.592,Z 487.964,A -85,B 0,C 180,E1 -19981.822,E2 -19981.822} C_VEL
LIN {X 0,Y 245.092,Z 497.734,A -85,B 0,C 180,E1 -19983.699,E2 -19983.699} C_VEL
LIN {X 0,Y 241.58,Z 506.473,A -85,B 0,C 180,E1 -19985.787,E2 -19985.787} C_VEL
LIN {X 0,Y 238.243,Z 514.104,A -85,B 0,C 180,E1 -19988.054,E2 -19988.054} C_VEL
LIN {X 0,Y 234.941,Z 521.258,A -85,B 0,C 180,E1 -19990.775,E2 -19990.775} C_VEL
LIN {X 0,Y 231.763,Z 527.626,A -85,B 0,C 180,E1 -19993.972,E2 -19993.972} C_VEL
LIN {X 0,Y 229.512,Z 531.826,A -85,B 0,C 180,E1 -19996.901,E2 -19996.901} C_VEL
LIN {X 0,Y 227.813,Z 534.764,A -85,B 0,C 180,E1 -19999.837,E2 -19999.837} C_VEL
LIN {X 0,Y 226.974,Z 536.09,A -85,B 0,C 180,E1 -20001.812,E2 -20001.812} C_VEL
LIN {X 0,Y 226.295,Z 536.936,A -85,B 0,C 180,E1 -20003.811,E2 -20003.811} C_VEL
LIN {X 0,Y 225.781,Z 537.259,A -85,B 0,C 180,E1 -20005.835,E2 -20005.835} C_VEL
LIN {X 0,Y 225.326,Z 536.734,A -85,B 0,C 180,E1 -20009.146,E2 -20009.146} C_VEL
LIN {X 0,Y 225.236,Z 534.694,A -85,B 0,C 180,E1 -20012.592,E2 -20012.592} C_VEL
LIN {X 0,Y 225.583,Z 531.273,A -85,B 0,C 180,E1 -20015.897,E2 -20015.897} C_VEL
LIN {X 0,Y 226.203,Z 526.557,A -85,B 0,C 180,E1 -20019.033,E2 -20019.033} C_VEL
LIN {X 0,Y 226.967,Z 520.579,A -85,B 0,C 180,E1 -20021.995,E2 -20021.995} C_VEL
LIN {X 0,Y 228.131,Z 513.142,A -85,B 0,C 180,E1 -20024.878,E2 -20024.878} C_VEL
LIN {X 0,Y 229.592,Z 503.953,A -85,B 0,C 180,E1 -20027.663,E2 -20027.663} C_VEL
LIN {X 0,Y 231.226,Z 494.485,A -85,B 0,C 180,E1 -20029.964,E2 -20029.964} C_VEL
LIN {X 0,Y 232.923,Z 483.545,A -85,B 0,C 180,E1 -20032.088,E2 -20032.088} C_VEL
LIN {X 0,Y 234.482,Z 473.308,A -85,B 0,C 180,E1 -20033.688,E2 -20033.688} C_VEL
LIN {X 0,Y 234.634,Z 471.319,A -85,B 0,C 180,E1 -20033.971,E2 -20033.971} C_VEL
LIN {X 0,Y 232.905,Z 458.465,A -85,B 0,C 180,E1 -20035.707,E2 -20035.707} C_VEL
LIN {X 0,Y 230.853,Z 445.681,A -85,B 0,C 180,E1 -20037.093,E2 -20037.093} C_VEL
LIN {X 0,Y 228.14,Z 431.347,A -85,B 0,C 180,E1 -20038.286,E2 -20038.286} C_VEL
LIN {X 0,Y 227.847,Z 429.673,A -85,B 0,C 180,E1 -20038.461,E2 -20038.461} C_VEL
LIN {X 0,Y 228.427,Z 422.951,A -85,B 0,C 180,E1 -20043.155,E2 -20043.155} C_VEL
LIN {X 0,Y 228.881,Z 417.341,A -85,B 0,C 180,E1 -20047.097,E2 -20047.097} C_VEL
LIN {X 0,Y 228.087,Z 412.201,A -85,B 0,C 180,E1 -20050.886,E2 -20050.886} C_VEL
LIN {X 0,Y 228.067,Z 412.077,A -85,B 0,C 180,E1 -20055.724,E2 -20055.724} C_VEL
LIN {X 0,Y 228.26,Z 412.053,A -85,B 0,C 180,E1 -20061.141,E2 -20061.141} C_VEL
LIN {X 0,Y 228.354,Z 412.327,A -85,B 0,C 180,E1 -20062.035,E2 -20062.035} C_VEL
LIN {X 0,Y 228.991,Z 416.403,A -85,B 0,C 180,E1 -20066.477,E2 -20066.477} C_VEL
LIN {X 0,Y 229.328,Z 418.064,A -85,B 0,C 180,E1 -20068.24,E2 -20068.24} C_VEL
LIN {X 0,Y 228.735,Z 421.692,A -85,B 0,C 180,E1 -20071.757,E2 -20071.757} C_VEL
LIN {X 0,Y 227.924,Z 427.342,A -85,B 0,C 180,E1 -20077.081,E2 -20077.081} C_VEL
LIN {X 0,Y 227.766,Z 428.767,A -85,B 0,C 180,E1 -20078.224,E2 -20078.224} C_VEL
LIN {X 0,Y 230.535,Z 441.095,A -85,B 0,C 180,E1 -20079.372,E2 -20079.372} C_VEL
LIN {X 0,Y 232.588,Z 452.609,A -85,B 0,C 180,E1 -20080.755,E2 -20080.755} C_VEL
LIN {X 0,Y 233.978,Z 463.456,A -85,B 0,C 180,E1 -20082.353,E2 -20082.353} C_VEL
LIN {X 0,Y 234.139,Z 467.405,A -85,B 0,C 180,E1 -20083.006,E2 -20083.006} C_VEL
LIN {X 0,Y 232.452,Z 477.797,A -85,B 0,C 180,E1 -20084.873,E2 -20084.873} C_VEL
LIN {X 0,Y 230.999,Z 486.239,A -85,B 0,C 180,E1 -20086.795,E2 -20086.795} C_VEL
LIN {X 0,Y 229.543,Z 494.132,A -85,B 0,C 180,E1 -20089.052,E2 -20089.052} C_VEL
LIN {X 0,Y 228.453,Z 500.122,A -85,B 0,C 180,E1 -20091.186,E2 -20091.186} C_VEL
LIN {X 0,Y 227.381,Z 505.677,A -85,B 0,C 180,E1 -20093.686,E2 -20093.686} C_VEL
LIN {X 0,Y 226.505,Z 510.794,A -85,B 0,C 180,E1 -20096.792,E2 -20096.792} C_VEL
LIN {X 0,Y 225.957,Z 514.13,A -85,B 0,C 180,E1 -20099.839,E2 -20099.839} C_VEL
LIN {X 0,Y 225.788,Z 516.019,A -85,B 0,C 180,E1 -20102.817,E2 -20102.817} C_VEL
LIN {X 0,Y 226.045,Z 516.531,A -85,B 0,C 180,E1 -20106.064,E2 -20106.064} C_VEL
LIN {X 0,Y 226.758,Z 515.559,A -85,B 0,C 180,E1 -20109.211,E2 -20109.211} C_VEL
LIN {X 0,Y 227.887,Z 513.181,A -85,B 0,C 180,E1 -20112.256,E2 -20112.256} C_VEL
LIN {X 0,Y 229.388,Z 509.416,A -85,B 0,C 180,E1 -20115.197,E2 -20115.197} C_VEL
LIN {X 0,Y 231.302,Z 504.203,A -85,B 0,C 180,E1 -20118.052,E2 -20118.052} C_VEL
LIN {X 0,Y 233.258,Z 498.428,A -85,B 0,C 180,E1 -20120.417,E2 -20120.417} C_VEL
LIN {X 0,Y 235.841,Z 490.714,A -85,B 0,C 180,E1 -20122.85,E2 -20122.85} C_VEL
LIN {X 0,Y 238.326,Z 482.243,A -85,B 0,C 180,E1 -20124.922,E2 -20124.922} C_VEL
LIN {X 0,Y 240.055,Z 475.825,A -85,B 0,C 180,E1 -20126.203,E2 -20126.203} C_VEL
LIN {X 0,Y 239.848,Z 467.511,A -85,B 0,C 180,E1 -20127.921,E2 -20127.921} C_VEL
LIN {X 0,Y 238.674,Z 458.274,A -85,B 0,C 180,E1 -20129.674,E2 -20129.674} C_VEL
LIN {X 0,Y 236.427,Z 448.861,A -85,B 0,C 180,E1 -20131.359,E2 -20131.359} C_VEL
LIN {X 0,Y 232.453,Z 437.304,A -85,B 0,C 180,E1 -20133.335,E2 -20133.335} C_VEL
LIN {X 0,Y 230.463,Z 432.689,A -85,B 0,C 180,E1 -20134.122,E2 -20134.122} C_VEL
LIN {X 0,Y 229.728,Z 430.247,A -85,B 0,C 180,E1 -20134.52,E2 -20134.52} C_VEL
LIN {X 0,Y 230.082,Z 428.447,A -85,B 0,C 180,E1 -20136.604,E2 -20136.604} C_VEL
LIN {X 0,Y 230.206,Z 426.903,A -85,B 0,C 180,E1 -20138.51,E2 -20138.51} C_VEL
LIN {X 0,Y 230.111,Z 424.104,A -85,B 0,C 180,E1 -20142.217,E2 -20142.217} C_VEL
LIN {X 0,Y 229.774,Z 421.693,A -85,B 0,C 180,E1 -20145.837,E2 -20145.837} C_VEL
LIN {X 0,Y 229.604,Z 419.491,A -85,B 0,C 180,E1 -20149.418,E2 -20149.418} C_VEL
LIN {X 0,Y 229.392,Z 417.567,A -85,B 0,C 180,E1 -20152.961,E2 -20152.961} C_VEL
LIN {X 0,Y 229.155,Z 415.209,A -85,B 0,C 180,E1 -20158.243,E2 -20158.243} C_VEL
LIN {X 0,Y 229.128,Z 414.558,A -85,B 0,C 180,E1 -20160.001,E2 -20160.001} C_VEL
LIN {X 0,Y 228.629,Z 413.632,A -85,B 0,C 180,E1 -20163.525,E2 -20163.525} C_VEL
LIN {X 0,Y 228.496,Z 412.913,A -85,B 0,C 180,E1 -20167.068,E2 -20167.068} C_VEL
LIN {X 0,Y 228.228,Z 412.57,A -85,B 0,C 180,E1 -20170.648,E2 -20170.648} C_VEL
LIN {X 0,Y 228.157,Z 412.67,A -85,B 0,C 180,E1 -20176.096,E2 -20176.096} C_VEL
LIN {X 0,Y 228.321,Z 413.635,A -85,B 0,C 180,E1 -20181.678,E2 -20181.678} C_VEL
LIN {X 0,Y 228.556,Z 414.79,A -85,B 0,C 180,E1 -20185.5,E2 -20185.5} C_VEL
LIN {X 0,Y 228.987,Z 417.109,A -85,B 0,C 180,E1 -20190.765,E2 -20190.765} C_VEL
LIN {X 0,Y 229.429,Z 419.069,A -85,B 0,C 180,E1 -20194.209,E2 -20194.209} C_VEL
LIN {X 0,Y 229.952,Z 421.845,A -85,B 0,C 180,E1 -20198.245,E2 -20198.245} C_VEL
LIN {X 0,Y 230.794,Z 425.743,A -85,B 0,C 180,E1 -20203.051,E2 -20203.051} C_VEL
LIN {X 0,Y 231.294,Z 428.141,A -85,B 0,C 180,E1 -20205.657,E2 -20205.657} C_VEL
LIN {X 0,Y 231.196,Z 429.124,A -85,B 0,C 180,E1 -20206.601,E2 -20206.601} C_VEL
LIN {X 0,Y 230.157,Z 430.864,A -85,B 0,C 180,E1 -20207.985,E2 -20207.985} C_VEL
LIN {X 0,Y 226.504,Z 435.33,A -85,B 0,C 180,E1 -20211.187,E2 -20211.187} C_VEL
LIN {X 0,Y 225.754,Z 437.162,A -85,B 0,C 180,E1 -20212.618,E2 -20212.618} C_VEL
LIN {X 0,Y 225.774,Z 437.732,A -85,B 0,C 180,E1 -20213.104,E2 -20213.104} C_VEL
LIN {X 0,Y 226.185,Z 439.93,A -85,B 0,C 180,E1 -20214.964,E2 -20214.964} C_VEL
LIN {X 0,Y 227.538,Z 443.425,A -85,B 0,C 180,E1 -20215.469,E2 -20215.469} C_VEL
LIN {X 0,Y 228.878,Z 447.135,A -85,B 0,C 180,E1 -20216.004,E2 -20216.004} C_VEL
LIN {X 0,Y 231.582,Z 459.347,A -85,B 0,C 180,E1 -20217.647,E2 -20217.647} C_VEL
LIN {X 0,Y 233.017,Z 470.61,A -85,B 0,C 180,E1 -20219.267,E2 -20219.267} C_VEL
LIN {X 0,Y 233.406,Z 481.191,A -85,B 0,C 180,E1 -20220.948,E2 -20220.948} C_VEL
LIN {X 0,Y 232.732,Z 491.843,A -85,B 0,C 180,E1 -20222.854,E2 -20222.854} C_VEL
LIN {X 0,Y 231.837,Z 497.301,A -85,B 0,C 180,E1 -20223.929,E2 -20223.929} C_VEL
LIN {X 0,Y 228.892,Z 506.874,A -85,B 0,C 180,E1 -20225.999,E2 -20225.999} C_VEL
LIN {X 0,Y 226.394,Z 514.668,A -85,B 0,C 180,E1 -20228.134,E2 -20228.134} C_VEL
LIN {X 0,Y 224.056,Z 522.223,A -85,B 0,C 180,E1 -20230.775,E2 -20230.775} C_VEL
LIN {X 0,Y 222.084,Z 528.274,A -85,B 0,C 180,E1 -20233.457,E2 -20233.457} C_VEL
LIN {X 0,Y 220.428,Z 533.042,A -85,B 0,C 180,E1 -20236.17,E2 -20236.17} C_VEL
LIN {X 0,Y 219.433,Z 536.681,A -85,B 0,C 180,E1 -20238.925,E2 -20238.925} C_VEL
LIN {X 0,Y 219.006,Z 538.524,A -85,B 0,C 180,E1 -20240.771,E2 -20240.771} C_VEL
LIN {X 0,Y 218.704,Z 540.451,A -85,B 0,C 180,E1 -20243.315,E2 -20243.315} C_VEL
LIN {X 0,Y 218.603,Z 544.266,A -85,B 0,C 180,E1 -20246.318,E2 -20246.318} C_VEL
LIN {X 0,Y 218.692,Z 545.973,A -85,B 0,C 180,E1 -20248.163,E2 -20248.163} C_VEL
LIN {X 0,Y 218.737,Z 547.24,A -85,B 0,C 180,E1 -20250.004,E2 -20250.004} C_VEL
LIN {X 0,Y 218.638,Z 548.091,A -85,B 0,C 180,E1 -20251.846,E2 -20251.846} C_VEL
LIN {X 0,Y 218.544,Z 548.57,A -85,B 0,C 180,E1 -20254.5,E2 -20254.5} C_VEL
LIN {X 0,Y 218.769,Z 548.169,A -85,B 0,C 180,E1 -20257.387,E2 -20257.387} C_VEL
LIN {X 0,Y 219.697,Z 546.288,A -85,B 0,C 180,E1 -20261.07,E2 -20261.07} C_VEL
LIN {X 0,Y 221.38,Z 542.753,A -85,B 0,C 180,E1 -20264.716,E2 -20264.716} C_VEL
LIN {X 0,Y 223.373,Z 539.01,A -85,B 0,C 180,E1 -20267.395,E2 -20267.395} C_VEL
LIN {X 0,Y 225.824,Z 534.229,A -85,B 0,C 180,E1 -20270.023,E2 -20270.023} C_VEL
LIN {X 0,Y 228.968,Z 527.421,A -85,B 0,C 180,E1 -20272.951,E2 -20272.951} C_VEL
LIN {X 0,Y 232.568,Z 519.653,A -85,B 0,C 180,E1 -20275.511,E2 -20275.511} C_VEL
LIN {X 0,Y 236.575,Z 510.476,A -85,B 0,C 180,E1 -20277.901,E2 -20277.901} C_VEL
LIN {X 0,Y 240.326,Z 501.175,A -85,B 0,C 180,E1 -20279.815,E2 -20279.815} C_VEL
LIN {X 0,Y 242.283,Z 491.045,A -85,B 0,C 180,E1 -20281.858,E2 -20281.858} C_VEL
LIN {X 0,Y 243.417,Z 480.295,A -85,B 0,C 180,E1 -20283.867,E2 -20283.867} C_VEL
LIN {X 0,Y 243.471,Z 470.045,A -85,B 0,C 180,E1 -20285.723,E2 -20285.723} C_VEL
LIN {X 0,Y 242.355,Z 461.097,A -85,B 0,C 180,E1 -20287.519,E2 -20287.519} C_VEL
LIN {X 0,Y 239.825,Z 455.01,A -85,B 0,C 180,E1 -20289.253,E2 -20289.253} C_VEL
LIN {X 0,Y 235.545,Z 446.134,A -85,B 0,C 180,E1 -20292.189,E2 -20292.189} C_VEL
LIN {X 0,Y 232.045,Z 440.076,A -85,B 0,C 180,E1 -20294.7,E2 -20294.7} C_VEL
LIN {X 0,Y 228.173,Z 434.385,A -85,B 0,C 180,E1 -20297.849,E2 -20297.849} C_VEL
LIN {X 0,Y 227.276,Z 431.857,A -85,B 0,C 180,E1 -20301.796,E2 -20301.796} C_VEL
LIN {X 0,Y 226.523,Z 430.321,A -85,B 0,C 180,E1 -20306.05,E2 -20306.05} C_VEL
LIN {X 0,Y 226.206,Z 429.769,A -85,B 0,C 180,E1 -20310.191,E2 -20310.191} C_VEL
LIN {X 0,Y 226.074,Z 430.127,A -85,B 0,C 180,E1 -20314.366,E2 -20314.366} C_VEL
LIN {X 0,Y 226.302,Z 431.277,A -85,B 0,C 180,E1 -20318.704,E2 -20318.704} C_VEL
LIN {X 0,Y 226.617,Z 432.932,A -85,B 0,C 180,E1 -20322.143,E2 -20322.143} C_VEL
LIN {X 0,Y 228.924,Z 436.779,A -85,B 0,C 180,E1 -20324.457,E2 -20324.457} C_VEL
LIN {X 0,Y 230.866,Z 438.947,A -85,B 0,C 180,E1 -20325.96,E2 -20325.96} C_VEL
LIN {X 0,Y 233.055,Z 442.838,A -85,B 0,C 180,E1 -20327.752,E2 -20327.752} C_VEL
LIN {X 0,Y 234.402,Z 444.675,A -85,B 0,C 180,E1 -20328.674,E2 -20328.674} C_VEL
LIN {X 0,Y 237.321,Z 450.331,A -85,B 0,C 180,E1 -20330.854,E2 -20330.854} C_VEL
LIN {X 0,Y 239.109,Z 454.623,A -85,B 0,C 180,E1 -20332.257,E2 -20332.257} C_VEL
LIN {X 0,Y 240.898,Z 461.656,A -85,B 0,C 180,E1 -20334.142,E2 -20334.142} C_VEL
LIN {X 0,Y 242.593,Z 471.841,A -85,B 0,C 180,E1 -20336.678,E2 -20336.678} C_VEL
LIN {X 0,Y 243.29,Z 480.167,A -85,B 0,C 180,E1 -20338.689,E2 -20338.689} C_VEL
LIN {X 0,Y 242.905,Z 489.145,A -85,B 0,C 180,E1 -20340.828,E2 -20340.828} C_VEL
LIN {X 0,Y 238.968,Z 499.655,A -85,B 0,C 180,E1 -20342.954,E2 -20342.954} C_VEL
LIN {X 0,Y 235.21,Z 508.327,A -85,B 0,C 180,E1 -20345.142,E2 -20345.142} C_VEL
LIN {X 0,Y 231.19,Z 516.716,A -85,B 0,C 180,E1 -20347.862,E2 -20347.862} C_VEL
LIN {X 0,Y 227.84,Z 523.365,A -85,B 0,C 180,E1 -20350.665,E2 -20350.665} C_VEL
LIN {X 0,Y 224.562,Z 529.294,A -85,B 0,C 180,E1 -20354.014,E2 -20354.014} C_VEL
LIN {X 0,Y 222.622,Z 532.528,A -85,B 0,C 180,E1 -20356.506,E2 -20356.506} C_VEL
LIN {X 0,Y 221.386,Z 534.508,A -85,B 0,C 180,E1 -20358.508,E2 -20358.508} C_VEL
LIN {X 0,Y 219.809,Z 536.698,A -85,B 0,C 180,E1 -20361.986,E2 -20361.986} C_VEL
LIN {X 0,Y 218.67,Z 537.497,A -85,B 0,C 180,E1 -20365.847,E2 -20365.847} C_VEL
LIN {X 0,Y 218.185,Z 536.583,A -85,B 0,C 180,E1 -20369.57,E2 -20369.57} C_VEL
LIN {X 0,Y 218.18,Z 534.159,A -85,B 0,C 180,E1 -20373.202,E2 -20373.202} C_VEL
LIN {X 0,Y 218.608,Z 530.47,A -85,B 0,C 180,E1 -20376.508,E2 -20376.508} C_VEL
LIN {X 0,Y 219.248,Z 525.459,A -85,B 0,C 180,E1 -20379.702,E2 -20379.702} C_VEL
LIN {X 0,Y 220.117,Z 519.166,A -85,B 0,C 180,E1 -20382.743,E2 -20382.743} C_VEL
LIN {X 0,Y 221.343,Z 511.324,A -85,B 0,C 180,E1 -20385.686,E2 -20385.686} C_VEL
LIN {X 0,Y 222.794,Z 502.874,A -85,B 0,C 180,E1 -20388.229,E2 -20388.229} C_VEL
LIN {X 0,Y 224.393,Z 493.658,A -85,B 0,C 180,E1 -20390.466,E2 -20390.466} C_VEL
LIN {X 0,Y 226.191,Z 482.474,A -85,B 0,C 180,E1 -20392.657,E2 -20392.657} C_VEL
LIN {X 0,Y 227.559,Z 473.587,A -85,B 0,C 180,E1 -20394.066,E2 -20394.066} C_VEL
LIN {X 0,Y 227.219,Z 468.592,A -85,B 0,C 180,E1 -20394.821,E2 -20394.821} C_VEL
LIN {X 0,Y 225.608,Z 456.625,A -85,B 0,C 180,E1 -20396.427,E2 -20396.427} C_VEL
LIN {X 0,Y 223.339,Z 442.679,A -85,B 0,C 180,E1 -20397.92,E2 -20397.92} C_VEL
LIN {X 0,Y 220.866,Z 429.844,A -85,B 0,C 180,E1 -20399.019,E2 -20399.019} C_VEL
LIN {X 0,Y 221.429,Z 423.383,A -85,B 0,C 180,E1 -20403.614,E2 -20403.614} C_VEL
LIN {X 0,Y 221.836,Z 419.014,A -85,B 0,C 180,E1 -20406.742,E2 -20406.742} C_VEL
LIN {X 0,Y 221.452,Z 415.22,A -85,B 0,C 180,E1 -20409.564,E2 -20409.564} C_VEL
LIN {X 0,Y 220.986,Z 412.959,A -85,B 0,C 180,E1 -20411.452,E2 -20411.452} C_VEL
LIN {X 0,Y 220.999,Z 412.958,A -85,B 0,C 180,E1 -20415.258,E2 -20415.258} C_VEL
LIN {X 0,Y 221.199,Z 412.933,A -85,B 0,C 180,E1 -20420.855,E2 -20420.855} C_VEL
LIN {X 0,Y 221.363,Z 413.438,A -85,B 0,C 180,E1 -20421.782,E2 -20421.782} C_VEL
LIN {X 0,Y 221.975,Z 417.547,A -85,B 0,C 180,E1 -20426.366,E2 -20426.366} C_VEL
LIN {X 0,Y 222.313,Z 419.208,A -85,B 0,C 180,E1 -20428.184,E2 -20428.184} C_VEL
LIN {X 0,Y 221.676,Z 422.862,A -85,B 0,C 180,E1 -20431.813,E2 -20431.813} C_VEL
LIN {X 0,Y 220.818,Z 428.757,A -85,B 0,C 180,E1 -20437.497,E2 -20437.497} C_VEL
LIN {X 0,Y 223.84,Z 442.519,A -85,B 0,C 180,E1 -20438.86,E2 -20438.86} C_VEL
LIN {X 0,Y 225.8,Z 453.564,A -85,B 0,C 180,E1 -20440.26,E2 -20440.26} C_VEL
LIN {X 0,Y 227.043,Z 463.803,A -85,B 0,C 180,E1 -20441.829,E2 -20441.829} C_VEL
LIN {X 0,Y 227.319,Z 467.643,A -85,B 0,C 180,E1 -20442.494,E2 -20442.494} C_VEL
LIN {X 0,Y 225.589,Z 478.106,A -85,B 0,C 180,E1 -20444.428,E2 -20444.428} C_VEL
LIN {X 0,Y 224.107,Z 486.492,A -85,B 0,C 180,E1 -20446.389,E2 -20446.389} C_VEL
LIN {X 0,Y 222.582,Z 494.357,A -85,B 0,C 180,E1 -20448.696,E2 -20448.696} C_VEL
LIN {X 0,Y 221.464,Z 500.411,A -85,B 0,C 180,E1 -20450.912,E2 -20450.912} C_VEL
LIN {X 0,Y 220.341,Z 505.995,A -85,B 0,C 180,E1 -20453.491,E2 -20453.491} C_VEL
LIN {X 0,Y 219.442,Z 511.051,A -85,B 0,C 180,E1 -20456.634,E2 -20456.634} C_VEL
LIN {X 0,Y 218.854,Z 514.534,A -85,B 0,C 180,E1 -20459.884,E2 -20459.884} C_VEL
LIN {X 0,Y 218.704,Z 516.546,A -85,B 0,C 180,E1 -20463.333,E2 -20463.333} C_VEL
LIN {X 0,Y 219.066,Z 516.932,A -85,B 0,C 180,E1 -20466.676,E2 -20466.676} C_VEL
LIN {X 0,Y 219.867,Z 515.803,A -85,B 0,C 180,E1 -20469.902,E2 -20469.902} C_VEL
LIN {X 0,Y 221.147,Z 513.31,A -85,B 0,C 180,E1 -20473.036,E2 -20473.036} C_VEL
LIN {X 0,Y 222.775,Z 509.408,A -85,B 0,C 180,E1 -20476.05,E2 -20476.05} C_VEL
LIN {X 0,Y 224.621,Z 504.713,A -85,B 0,C 180,E1 -20478.662,E2 -20478.662} C_VEL
LIN {X 0,Y 226.959,Z 498.23,A -85,B 0,C 180,E1 -20481.359,E2 -20481.359} C_VEL
LIN {X 0,Y 229.361,Z 491.452,A -85,B 0,C 180,E1 -20483.538,E2 -20483.538} C_VEL
LIN {X 0,Y 231.955,Z 483.179,A -85,B 0,C 180,E1 -20485.645,E2 -20485.645} C_VEL
LIN {X 0,Y 233.758,Z 476.777,A -85,B 0,C 180,E1 -20486.981,E2 -20486.981} C_VEL
LIN {X 0,Y 233.403,Z 466.426,A -85,B 0,C 180,E1 -20489.211,E2 -20489.211} C_VEL
LIN {X 0,Y 232.016,Z 457.35,A -85,B 0,C 180,E1 -20491.011,E2 -20491.011} C_VEL
LIN {X 0,Y 229.39,Z 447.449,A -85,B 0,C 180,E1 -20492.895,E2 -20492.895} C_VEL
LIN {X 0,Y 225.789,Z 437.519,A -85,B 0,C 180,E1 -20494.723,E2 -20494.723} C_VEL
LIN {X 0,Y 224.185,Z 433.923,A -85,B 0,C 180,E1 -20495.396,E2 -20495.396} C_VEL
LIN {X 0,Y 223.003,Z 430.589,A -85,B 0,C 180,E1 -20495.98,E2 -20495.98} C_VEL
LIN {X 0,Y 223.211,Z 429.117,A -85,B 0,C 180,E1 -20497.801,E2 -20497.801} C_VEL
LIN {X 0,Y 223.274,Z 426.231,A -85,B 0,C 180,E1 -20501.654,E2 -20501.654} C_VEL
LIN {X 0,Y 222.927,Z 423.795,A -85,B 0,C 180,E1 -20505.392,E2 -20505.392} C_VEL
LIN {X 0,Y 222.771,Z 421.592,A -85,B 0,C 180,E1 -20509.089,E2 -20509.089} C_VEL
LIN {X 0,Y 222.581,Z 419.675,A -85,B 0,C 180,E1 -20512.745,E2 -20512.745} C_VEL
LIN {X 0,Y 222.376,Z 417.321,A -85,B 0,C 180,E1 -20518.19,E2 -20518.19} C_VEL
LIN {X 0,Y 222.353,Z 416.67,A -85,B 0,C 180,E1 -20520.001,E2 -20520.001} C_VEL
LIN {X 0,Y 221.87,Z 415.77,A -85,B 0,C 180,E1 -20523.633,E2 -20523.633} C_VEL
LIN {X 0,Y 221.743,Z 415.094,A -85,B 0,C 180,E1 -20527.284,E2 -20527.284} C_VEL
LIN {X 0,Y 221.475,Z 414.816,A -85,B 0,C 180,E1 -20530.977,E2 -20530.977} C_VEL
LIN {X 0,Y 221.445,Z 415.004,A -85,B 0,C 180,E1 -20536.597,E2 -20536.597} C_VEL
LIN {X 0,Y 221.634,Z 416.092,A -85,B 0,C 180,E1 -20542.367,E2 -20542.367} C_VEL
LIN {X 0,Y 221.939,Z 417.855,A -85,B 0,C 180,E1 -20547.555,E2 -20547.555} C_VEL
LIN {X 0,Y 222.445,Z 420.255,A -85,B 0,C 180,E1 -20552.487,E2 -20552.487} C_VEL
LIN {X 0,Y 222.971,Z 422.924,A -85,B 0,C 180,E1 -20556.79,E2 -20556.79} C_VEL
LIN {X 0,Y 223.641,Z 426.287,A -85,B 0,C 180,E1 -20561.296,E2 -20561.296} C_VEL
LIN {X 0,Y 224.445,Z 430.031,A -85,B 0,C 180,E1 -20565.632,E2 -20565.632} C_VEL
LIN {X 0,Y 225.249,Z 434.599,A -85,B 0,C 180,E1 -20570.244,E2 -20570.244} C_VEL
LIN {X 0,Y 225.774,Z 437.732,A -85,B 0,C 180,E1 -20573.104,E2 -20573.104} C_VEL
LIN {X 0,Y 226.002,Z 439.472,A -85,B 0,C 180,E1 -20573.96,E2 -20573.96} C_VEL
LIN {X 0,Y 226.238,Z 442.152,A -85,B 0,C 180,E1 -20574.656,E2 -20574.656} C_VEL
LIN {X 0,Y 226.461,Z 447.199,A -85,B 0,C 180,E1 -20575.449,E2 -20575.449} C_VEL
LIN {X 0,Y 226.264,Z 461.109,A -85,B 0,C 180,E1 -20576.809,E2 -20576.809} C_VEL
LIN {X 0,Y 226.279,Z 464.944,A -85,B 0,C 180,E1 -20577.292,E2 -20577.292} C_VEL
